C03640=1088.858,407.199,-100.671,177.784,26.140,154.193
C03641=1088.865,407.445,-100.711,177.788,26.148,154.195
C03642=1088.871,407.692,-100.752,177.791,26.157,154.197
C03643=1088.878,407.938,-100.792,177.795,26.166,154.199
C03644=1088.884,408.185,-100.832,177.797,26.175,154.200
C03645=1088.890,408.432,-100.873,177.800,26.183,154.202
C03646=1088.896,408.678,-100.913,177.804,26.192,154.204
C03647=1088.903,408.925,-100.953,177.807,26.201,154.206
C03648=1088.909,409.172,-100.994,177.811,26.210,154.207
C03649=1088.915,409.419,-101.034,177.815,26.219,154.209
C03650=1088.922,409.665,-101.075,177.818,26.227,154.211
C03651=1088.927,409.911,-101.116,177.821,26.236,154.213
C03652=1088.934,410.158,-101.156,177.824,26.245,154.215
C03653=1088.940,410.404,-101.196,177.828,26.254,154.217
C03654=1088.946,410.652,-101.237,177.831,26.263,154.218
C03655=1088.953,410.879,-101.274,177.834,26.272,154.220
C03656=1088.958,411.106,-101.312,177.837,26.280,154.222
C03657=1088.963,411.333,-101.349,177.841,26.288,154.223
C03658=1088.969,411.560,-101.387,177.844,26.297,154.225
C03659=1088.976,411.787,-101.425,177.847,26.305,154.227
C03660=1088.981,412.014,-101.462,177.850,26.313,154.228
C03661=1088.987,412.241,-101.500,177.852,26.322,154.230
C03662=1088.993,412.469,-101.537,177.855,26.330,154.232
C03663=1089.000,412.716,-101.578,177.859,26.339,154.234
C03664=1089.006,412.962,-101.619,177.863,26.349,154.236
C03665=1089.012,413.209,-101.660,177.866,26.358,154.238
C03666=1089.019,413.455,-101.701,177.869,26.368,154.240
C03667=1089.025,413.702,-101.742,177.873,26.377,154.241
C03668=1089.032,413.948,-101.782,177.876,26.386,154.243
C03669=1089.038,414.195,-101.824,177.880,26.395,154.245
C03670=1089.045,414.441,-101.864,177.883,26.405,154.247
C03671=1089.051,414.688,-101.906,177.886,26.414,154.249
C03672=1089.058,414.934,-101.947,177.890,26.423,154.251
C03673=1089.063,415.181,-101.988,177.894,26.433,154.253
C03674=1089.071,415.428,-102.029,177.896,26.442,154.255
C03675=1089.077,415.674,-102.070,177.900,26.452,154.257
C03676=1089.084,415.921,-102.111,177.904,26.462,154.259
C03677=1089.090,416.167,-102.152,177.908,26.471,154.261
C03678=1089.096,416.413,-102.194,177.910,26.481,154.263
C03679=1089.103,416.660,-102.235,177.914,26.490,154.265
C03680=1089.109,416.906,-102.277,177.918,26.500,154.267
C03681=1089.115,417.153,-102.318,177.921,26.510,154.269
C03682=1089.122,417.399,-102.359,177.924,26.520,154.271
C03683=1089.128,417.645,-102.401,177.928,26.529,154.273
C03684=1089.135,417.892,-102.443,177.931,26.539,154.275
C03685=1089.140,418.138,-102.484,177.935,26.549,154.277
C03686=1089.148,418.385,-102.525,177.939,26.559,154.279
C03687=1089.154,418.631,-102.567,177.941,26.569,154.281
C03688=1089.160,418.878,-102.609,177.945,26.579,154.283
C03689=1089.166,419.124,-102.650,177.949,26.589,154.285
C03690=1089.173,419.371,-102.692,177.952,26.599,154.288
C03691=1089.179,419.617,-102.733,177.956,26.609,154.290
C03692=1089.186,419.864,-102.774,177.960,26.619,154.292
C03693=1089.192,420.110,-102.817,177.963,26.630,154.294
C03694=1089.199,420.356,-102.858,177.966,26.639,154.296
C03695=1089.205,420.603,-102.900,177.970,26.649,154.298
C03696=1089.211,420.850,-102.942,177.973,26.660,154.300
C03697=1089.219,421.096,-102.984,177.977,26.670,154.302
C03698=1089.225,421.342,-103.025,177.980,26.680,154.305
C03699=1089.231,421.589,-103.067,177.984,26.691,154.307
C03700=1089.238,421.834,-103.109,177.988,26.701,154.309
C03701=1089.244,422.081,-103.151,177.991,26.711,154.311
C03702=1089.251,422.327,-103.194,177.995,26.722,154.313
C03703=1089.257,422.574,-103.235,177.998,26.732,154.316
C03704=1089.264,422.820,-103.278,178.002,26.743,154.318
C03705=1089.270,423.067,-103.319,178.006,26.753,154.320
C03706=1089.277,423.312,-103.362,178.009,26.764,154.322
C03707=1089.283,423.559,-103.403,178.013,26.775,154.324
C03708=1089.290,423.806,-103.446,178.016,26.785,154.327
C03709=1089.296,424.051,-103.488,178.020,26.796,154.329
C03710=1089.303,424.298,-103.530,178.023,26.807,154.331
C03711=1089.311,424.618,-103.585,178.027,26.820,154.334
C03712=1089.319,424.939,-103.640,178.032,26.834,154.337
C03713=1089.328,425.259,-103.695,178.037,26.849,154.340
C03714=1089.336,425.580,-103.750,178.042,26.863,154.343
C03715=1089.343,425.825,-103.793,178.045,26.874,154.346
C03716=1089.349,426.071,-103.835,178.049,26.884,154.348
C03717=1089.356,426.318,-103.878,178.052,26.895,154.350
C03718=1089.363,426.564,-103.920,178.056,26.906,154.353
C03719=1089.369,426.811,-103.963,178.059,26.918,154.355
C03720=1089.376,427.056,-104.006,178.063,26.928,154.357
C03721=1089.382,427.302,-104.048,178.067,26.940,154.360
C03722=1089.389,427.549,-104.091,178.071,26.951,154.362
C03723=1089.396,427.795,-104.133,178.074,26.962,154.365
C03724=1089.402,428.042,-104.176,178.078,26.973,154.367
C03725=1089.409,428.288,-104.219,178.081,26.985,154.369
C03726=1089.415,428.533,-104.261,178.085,26.996,154.372
C03727=1089.422,428.780,-104.304,178.088,27.007,154.374
C03728=1089.429,429.026,-104.347,178.093,27.019,154.377
C03729=1089.436,429.272,-104.390,178.096,27.030,154.379
C03730=1089.442,429.518,-104.432,178.100,27.041,154.382
C03731=1089.448,429.765,-104.476,178.103,27.053,154.384
C03732=1089.456,430.011,-104.519,178.107,27.065,154.387
C03733=1089.462,430.257,-104.562,178.111,27.076,154.389
C03734=1089.469,430.503,-104.605,178.115,27.088,154.392
C03735=1089.474,430.749,-104.648,178.118,27.099,154.394
C03736=1089.481,430.995,-104.691,178.121,27.111,154.397
C03737=1089.488,431.241,-104.734,178.125,27.123,154.399
C03738=1089.495,431.487,-104.777,178.129,27.135,154.402
C03739=1089.502,431.733,-104.820,178.133,27.146,154.404
C03740=1089.508,431.979,-104.863,178.136,27.158,154.407
C03741=1089.515,432.225,-104.907,178.141,27.171,154.410
C03742=1089.521,432.472,-104.950,178.144,27.182,154.412
C03743=1089.528,432.717,-104.993,178.147,27.194,154.415
C03744=1089.535,432.963,-105.037,178.151,27.206,154.418
C03745=1089.542,433.210,-105.079,178.155,27.218,154.420
C03746=1089.548,433.456,-105.123,178.159,27.231,154.423
C03747=1089.554,433.702,-105.167,178.162,27.242,154.426
C03748=1089.562,433.947,-105.210,178.166,27.255,154.428
C03749=1089.568,434.194,-105.253,178.170,27.267,154.431
C03750=1089.575,434.441,-105.298,178.173,27.279,154.434
C03751=1089.586,434.835,-105.368,178.180,27.300,154.438
C03752=1089.596,435.230,-105.438,178.186,27.319,154.442
C03753=1089.607,435.626,-105.508,178.192,27.339,154.447
C03754=1089.617,436.021,-105.578,178.198,27.359,154.451
C03755=1089.624,436.266,-105.622,178.202,27.372,154.454
C03756=1089.631,436.512,-105.666,178.205,27.385,154.457
C03757=1089.638,436.759,-105.710,178.209,27.398,154.460
C03758=1089.645,437.004,-105.754,178.213,27.410,154.463
C03759=1089.651,437.250,-105.798,178.217,27.423,154.465
C03760=1089.658,437.496,-105.841,178.220,27.436,154.468
C03761=1089.664,437.742,-105.886,178.225,27.449,154.471
C03762=1089.671,437.988,-105.930,178.228,27.461,154.474
C03763=1089.680,438.310,-105.987,178.234,27.479,154.478
C03764=1089.689,438.630,-106.045,178.238,27.495,154.481
C03765=1089.698,438.952,-106.103,178.244,27.512,154.485
C03766=1089.707,439.273,-106.161,178.248,27.529,154.489
C03767=1089.714,439.519,-106.204,178.252,27.543,154.492
C03768=1089.720,439.764,-106.249,178.256,27.556,154.495
C03769=1089.728,440.010,-106.293,178.260,27.569,154.498
C03770=1089.735,440.256,-106.337,178.264,27.583,154.501
C03771=1089.742,440.501,-106.382,178.268,27.596,154.504
C03772=1089.748,440.748,-106.426,178.272,27.609,154.507
C03773=1089.755,440.993,-106.471,178.275,27.623,154.510
C03774=1089.762,441.240,-106.515,178.279,27.637,154.513
C03775=1089.768,441.485,-106.560,178.284,27.650,154.516
C03776=1089.775,441.731,-106.604,178.287,27.664,154.519
C03777=1089.782,441.977,-106.649,178.291,27.677,154.522
C03778=1089.789,442.222,-106.694,178.296,27.691,154.525
C03779=1089.797,442.468,-106.739,178.299,27.705,154.529
C03780=1089.803,442.714,-106.783,178.303,27.719,154.532
C03781=1089.810,442.959,-106.827,178.307,27.733,154.535
C03782=1089.816,443.206,-106.873,178.311,27.747,154.538
C03783=1089.823,443.451,-106.917,178.315,27.761,154.541
C03784=1089.830,443.697,-106.962,178.319,27.775,154.544
C03785=1089.837,443.943,-107.007,178.323,27.789,154.547
C03786=1089.844,444.189,-107.052,178.327,27.803,154.551
C03787=1089.851,444.434,-107.098,178.331,27.817,154.554
C03788=1089.858,444.680,-107.143,178.335,27.832,154.557
C03789=1089.865,444.925,-107.187,178.338,27.846,154.560
C03790=1089.872,445.171,-107.232,178.342,27.860,154.564
C03791=1089.879,445.418,-107.278,178.345,27.874,154.567
C03792=1089.886,445.662,-107.323,178.348,27.888,154.570
C03793=1089.893,445.908,-107.368,178.351,27.903,154.574
C03794=1089.899,446.154,-107.413,178.354,27.917,154.577
C03795=1089.907,446.399,-107.459,178.356,27.931,154.580
C03796=1089.913,446.646,-107.504,178.358,27.945,154.584
C03797=1089.920,446.891,-107.549,178.361,27.959,154.587
C03798=1089.928,447.137,-107.594,178.363,27.973,154.591
C03799=1089.934,447.383,-107.640,178.364,27.987,154.594
C03800=1089.941,447.628,-107.685,178.366,28.001,154.597
C03801=1089.948,447.874,-107.731,178.367,28.015,154.601
C03802=1089.956,448.119,-107.776,178.368,28.030,154.604
C03803=1089.962,448.366,-107.822,178.370,28.043,154.608
C03804=1089.969,448.611,-107.867,178.371,28.058,154.611
C03805=1089.976,448.857,-107.913,178.372,28.071,154.615
C03806=1089.983,449.102,-107.958,178.373,28.086,154.618
C03807=1089.990,449.347,-108.004,178.373,28.100,154.622
C03808=1089.997,449.593,-108.050,178.374,28.114,154.625
C03809=1090.004,449.838,-108.094,178.374,28.128,154.629
C03810=1090.015,450.084,-108.139,178.374,28.140,154.632
C03811=1089.633,450.077,-108.327,178.332,28.336,154.686
C03812=1089.623,449.830,-108.284,178.331,28.323,154.682
C03813=1089.615,449.585,-108.238,178.330,28.310,154.679
C03814=1089.609,449.340,-108.192,178.330,28.295,154.675
C03815=1089.602,449.095,-108.147,178.329,28.281,154.672
C03816=1089.594,448.849,-108.102,178.329,28.267,154.669
C03817=1089.587,448.603,-108.056,178.327,28.253,154.665
C03818=1089.580,448.358,-108.010,178.326,28.239,154.662
C03819=1089.573,448.111,-107.964,178.325,28.225,154.658
C03820=1089.566,447.867,-107.919,178.324,28.211,154.655
C03821=1089.559,447.620,-107.874,178.322,28.197,154.651
C03822=1089.552,447.375,-107.828,178.320,28.183,154.648
C03823=1089.545,447.128,-107.782,178.318,28.169,154.644
C03824=1089.538,446.884,-107.737,178.316,28.154,154.641
C03825=1089.532,446.637,-107.692,178.314,28.140,154.637
C03826=1089.524,446.392,-107.646,178.311,28.126,154.634
C03827=1089.517,446.146,-107.601,178.309,28.111,154.631
C03828=1089.510,445.901,-107.555,178.306,28.097,154.627
C03829=1089.503,445.655,-107.510,178.303,28.083,154.624
C03830=1089.497,445.409,-107.465,178.300,28.069,154.621
C03831=1089.489,445.164,-107.419,178.296,28.055,154.617
C03832=1089.482,444.918,-107.374,178.293,28.040,154.614
C03833=1089.475,444.672,-107.330,178.289,28.027,154.611
C03834=1089.468,444.426,-107.284,178.285,28.012,154.607
C03835=1089.462,444.181,-107.239,178.281,27.998,154.604
C03836=1089.454,443.935,-107.194,178.277,27.984,154.601
C03837=1089.448,443.690,-107.150,178.273,27.969,154.598
C03838=1089.441,443.443,-107.104,178.269,27.955,154.595
C03839=1089.434,443.198,-107.060,178.264,27.941,154.591
C03840=1089.427,442.952,-107.015,178.261,27.927,154.588
C03841=1089.420,442.707,-106.970,178.257,27.913,154.585
C03842=1089.413,442.460,-106.925,178.252,27.899,154.582
C03843=1089.406,442.215,-106.881,178.249,27.886,154.579
C03844=1089.400,441.969,-106.835,178.245,27.872,154.576
C03845=1089.393,441.723,-106.790,178.240,27.858,154.573
C03846=1089.385,441.477,-106.745,178.237,27.844,154.570
C03847=1089.379,441.232,-106.701,178.233,27.831,154.567
C03848=1089.372,440.986,-106.657,178.229,27.817,154.563
C03849=1089.365,440.740,-106.612,178.225,27.803,154.560
C03850=1089.358,440.495,-106.568,178.220,27.790,154.557
C03851=1089.351,440.249,-106.523,178.217,27.777,154.554
C03852=1089.345,440.003,-106.479,178.213,27.763,154.551
C03853=1089.338,439.757,-106.434,178.209,27.750,154.548
C03854=1089.331,439.511,-106.390,178.205,27.736,154.545
C03855=1089.324,439.265,-106.345,178.201,27.723,154.542
C03856=1089.315,438.957,-106.290,178.196,27.707,154.539
C03857=1089.307,438.648,-106.235,178.191,27.690,154.535
C03858=1089.298,438.340,-106.179,178.186,27.674,154.531
C03859=1089.290,438.031,-106.124,178.181,27.658,154.528
C03860=1089.283,437.785,-106.080,178.177,27.645,154.525
C03861=1089.275,437.540,-106.036,178.174,27.632,154.522
C03862=1089.269,437.294,-105.992,178.169,27.619,154.519
C03863=1089.262,437.048,-105.948,178.166,27.606,154.516
C03864=1089.255,436.801,-105.904,178.162,27.593,154.514
C03865=1089.249,436.556,-105.859,178.158,27.581,154.511
C03866=1089.241,436.310,-105.816,178.154,27.568,154.508
C03867=1089.235,436.064,-105.772,178.150,27.555,154.505
C03868=1089.229,435.818,-105.728,178.146,27.543,154.502
C03869=1089.222,435.572,-105.684,178.142,27.530,154.500
C03870=1089.214,435.326,-105.641,178.139,27.518,154.497
C03871=1089.208,435.080,-105.597,178.135,27.505,154.494
C03872=1089.202,434.834,-105.553,178.131,27.493,154.491
C03873=1089.195,434.588,-105.509,178.127,27.480,154.489
C03874=1089.188,434.342,-105.466,178.124,27.468,154.486
C03875=1089.181,434.096,-105.422,178.119,27.456,154.483
C03876=1089.175,433.850,-105.378,178.116,27.443,154.480
C03877=1089.168,433.605,-105.335,178.112,27.431,154.478
C03878=1089.161,433.359,-105.291,178.108,27.419,154.475
C03879=1089.155,433.112,-105.248,178.104,27.407,154.472
C03880=1089.149,432.866,-105.204,178.101,27.394,154.470
C03881=1089.141,432.620,-105.160,178.096,27.382,154.467
C03882=1089.135,432.373,-105.117,178.093,27.371,154.464
C03883=1089.128,432.127,-105.074,178.089,27.358,154.462
C03884=1089.121,431.882,-105.030,178.085,27.346,154.459
C03885=1089.115,431.635,-104.988,178.081,27.335,154.457
C03886=1089.108,431.389,-104.944,178.078,27.323,154.454
C03887=1089.101,431.143,-104.901,178.074,27.311,154.451
C03888=1089.094,430.897,-104.858,178.071,27.299,154.449
C03889=1089.088,430.651,-104.815,178.066,27.287,154.446
C03890=1089.081,430.405,-104.772,178.063,27.276,154.444
C03891=1089.075,430.158,-104.729,178.059,27.264,154.441
C03892=1089.068,429.913,-104.685,178.056,27.253,154.439
C03893=1089.062,429.667,-104.643,178.051,27.241,154.436
C03894=1089.055,429.421,-104.600,178.048,27.230,154.434
C03895=1089.048,429.175,-104.557,178.044,27.218,154.431
C03896=1089.042,428.928,-104.514,178.041,27.206,154.429
C03897=1089.035,428.682,-104.471,178.037,27.195,154.426
C03898=1089.028,428.436,-104.428,178.033,27.184,154.424
C03899=1089.022,428.190,-104.385,178.030,27.172,154.421
C03900=1089.015,427.944,-104.342,178.025,27.161,154.419
C03901=1089.008,427.697,-104.300,178.022,27.150,154.417
C03902=1089.001,427.451,-104.257,178.018,27.139,154.414
C03903=1088.996,427.205,-104.214,178.015,27.128,154.412
C03904=1088.989,426.959,-104.172,178.011,27.116,154.409
C03905=1088.982,426.713,-104.129,178.007,27.106,154.407
C03906=1088.975,426.466,-104.087,178.004,27.094,154.405
C03907=1088.968,426.220,-104.044,178.000,27.083,154.402
C03908=1088.962,425.984,-104.004,177.996,27.073,154.400
C03909=1088.956,425.750,-103.963,177.993,27.062,154.398
C03910=1088.950,425.514,-103.922,177.989,27.052,154.396
C03911=1088.944,425.279,-103.882,177.986,27.042,154.393
C03912=1088.937,425.044,-103.841,177.983,27.031,154.391
C03913=1088.931,424.809,-103.801,177.979,27.021,154.389
C03914=1088.925,424.572,-103.760,177.975,27.010,154.387
C03915=1088.919,424.337,-103.719,177.972,27.000,154.384
C03916=1088.912,424.091,-103.677,177.969,26.989,154.382
C03917=1088.906,423.845,-103.635,177.965,26.979,154.380
C03918=1088.899,423.598,-103.593,177.962,26.968,154.378
C03919=1088.893,423.353,-103.551,177.958,26.958,154.375
C03920=1088.886,423.106,-103.508,177.954,26.947,154.373
C03921=1088.879,422.859,-103.466,177.951,26.936,154.371
C03922=1088.873,422.614,-103.424,177.947,26.925,154.369
C03923=1088.867,422.367,-103.382,177.943,26.915,154.366
C03924=1088.860,422.121,-103.340,177.940,26.904,154.364
C03925=1088.854,421.874,-103.298,177.936,26.894,154.362
C03926=1088.847,421.628,-103.256,177.932,26.884,154.360
C03927=1088.840,421.381,-103.214,177.929,26.873,154.358
C03928=1088.834,421.136,-103.172,177.925,26.863,154.355
C03929=1088.828,420.889,-103.130,177.921,26.853,154.353
C03930=1088.821,420.643,-103.089,177.918,26.843,154.351
C03931=1088.814,420.397,-103.047,177.915,26.832,154.349
C03932=1088.807,420.150,-103.005,177.911,26.822,154.347
C03933=1088.802,419.903,-102.963,177.907,26.812,154.345
C03934=1088.795,419.657,-102.921,177.904,26.802,154.343
C03935=1088.789,419.411,-102.879,177.900,26.792,154.341
C03936=1088.781,419.164,-102.838,177.896,26.781,154.338
C03937=1088.775,418.918,-102.797,177.894,26.772,154.336
C03938=1088.769,418.671,-102.755,177.890,26.762,154.334
C03939=1088.763,418.425,-102.713,177.886,26.752,154.332
C03940=1088.756,418.178,-102.672,177.882,26.742,154.330
C03941=1088.750,417.932,-102.631,177.879,26.732,154.328
C03942=1088.743,417.685,-102.589,177.876,26.722,154.326
C03943=1088.737,417.439,-102.547,177.872,26.712,154.324
C03944=1088.730,417.181,-102.503,177.869,26.702,154.322
C03945=1088.723,416.924,-102.461,177.865,26.691,154.320
C03946=1088.717,416.666,-102.417,177.861,26.681,154.317
C03947=1088.710,416.408,-102.373,177.858,26.671,154.315
C03948=1088.704,416.162,-102.332,177.854,26.661,154.313
C03949=1088.698,415.915,-102.292,177.850,26.652,154.311
C03950=1088.691,415.669,-102.250,177.847,26.643,154.309
C03951=1088.684,415.423,-102.209,177.844,26.633,154.307
C03952=1088.678,415.176,-102.167,177.840,26.623,154.305
C03953=1088.671,414.930,-102.126,177.837,26.614,154.303
C03954=1088.665,414.682,-102.085,177.833,26.604,154.301
C03955=1088.658,414.436,-102.044,177.829,26.595,154.300
C03956=1088.652,414.190,-102.002,177.826,26.585,154.298
C03957=1088.645,413.943,-101.962,177.823,26.576,154.296
C03958=1088.639,413.697,-101.921,177.819,26.567,154.294
C03959=1088.632,413.450,-101.880,177.816,26.557,154.292
C03960=1088.626,413.204,-101.839,177.812,26.548,154.290
C03961=1088.620,412.957,-101.798,177.809,26.539,154.288
C03962=1088.613,412.710,-101.757,177.806,26.530,154.286
C03963=1088.607,412.464,-101.716,177.802,26.520,154.284
C03964=1088.602,412.241,-101.680,177.799,26.512,154.283
C03965=1088.595,412.020,-101.643,177.796,26.504,154.281
C03966=1088.589,411.798,-101.606,177.793,26.495,154.279
C03967=1088.584,411.575,-101.570,177.790,26.487,154.278
C03968=1088.578,411.353,-101.533,177.787,26.479,154.276
C03969=1088.572,411.131,-101.496,177.784,26.471,154.274
C03970=1088.567,410.909,-101.460,177.780,26.463,154.273
C03971=1088.561,410.687,-101.422,177.777,26.455,154.271
C03972=1088.555,410.440,-101.382,177.774,26.445,154.269
C03973=1088.548,410.194,-101.341,177.771,26.437,154.267
C03974=1088.542,409.948,-101.301,177.767,26.427,154.265
C03975=1088.535,409.700,-101.260,177.764,26.419,154.264
C03976=1088.529,409.454,-101.220,177.760,26.410,154.262
C03977=1088.523,409.207,-101.179,177.757,26.401,154.260
C03978=1088.517,408.961,-101.138,177.753,26.392,154.258
C03979=1088.510,408.715,-101.098,177.750,26.383,154.256
C03980=1088.505,408.468,-101.057,177.747,26.374,154.255
C03981=1088.498,408.221,-101.017,177.744,26.365,154.253
C03982=1088.492,407.975,-100.977,177.740,26.357,154.251
C03983=1088.486,407.727,-100.936,177.737,26.348,154.249
C03984=1088.479,407.481,-100.896,177.733,26.339,154.247
C03985=1088.473,407.234,-100.856,177.730,26.331,154.246
C03986=1088.467,406.988,-100.816,177.726,26.321,154.244
C03987=1088.460,406.741,-100.775,177.723,26.313,154.242
C03988=1088.455,406.494,-100.735,177.720,26.305,154.241
C03989=1088.448,406.248,-100.695,177.716,26.296,154.239
C03990=1088.442,406.001,-100.654,177.713,26.288,154.237
C03991=1088.435,405.755,-100.614,177.710,26.278,154.235
C03992=1088.429,405.508,-100.575,177.707,26.271,154.234
C03993=1088.423,405.261,-100.535,177.704,26.262,154.232
C03994=1088.416,405.014,-100.494,177.700,26.254,154.230
C03995=1088.410,404.767,-100.454,177.697,26.245,154.229
C03996=1088.403,404.520,-100.415,177.693,26.236,154.227
C03997=1088.397,404.274,-100.374,177.690,26.228,154.225
C03998=1088.391,404.027,-100.334,177.687,26.220,154.224
C03999=1088.384,403.781,-100.294,177.683,26.211,154.222
C04000=1088.378,403.534,-100.255,177.680,26.203,154.220
C04001=1088.372,403.287,-100.215,177.677,26.195,154.219
C04002=1088.366,403.040,-100.175,177.673,26.187,154.217
C04003=1088.359,402.794,-100.135,177.670,26.178,154.215
C04004=1088.353,402.547,-100.095,177.667,26.171,154.214
C04005=1088.347,402.300,-100.055,177.663,26.162,154.212
C04006=1088.341,402.054,-100.016,177.660,26.154,154.211
C04007=1088.335,401.807,-99.976,177.657,26.146,154.209
C04008=1088.329,401.560,-99.936,177.653,26.138,154.207
C04009=1088.322,401.314,-99.897,177.650,26.130,154.206
C04010=1088.316,401.066,-99.858,177.647,26.122,154.204
C04011=1088.309,400.820,-99.818,177.644,26.114,154.203
C04012=1088.303,400.573,-99.778,177.640,26.106,154.201
C04013=1088.297,400.326,-99.738,177.637,26.098,154.200
C04014=1088.291,400.079,-99.699,177.634,26.090,154.198
C04015=1088.285,399.833,-99.660,177.631,26.082,154.196
C04016=1088.278,399.587,-99.620,177.627,26.074,154.195
C04017=1088.272,399.339,-99.581,177.624,26.066,154.193
C04018=1088.266,399.092,-99.541,177.621,26.058,154.192
C04019=1088.260,398.845,-99.502,177.618,26.050,154.190
C04020=1088.255,398.618,-99.466,177.615,26.043,154.189
C04021=1088.249,398.392,-99.429,177.611,26.036,154.187
C04022=1088.243,398.164,-99.393,177.608,26.029,154.186
C04023=1088.237,397.938,-99.357,177.606,26.022,154.185
C04024=1088.231,397.711,-99.321,177.603,26.015,154.183
C04025=1088.225,397.483,-99.285,177.600,26.007,154.182
C04026=1088.220,397.256,-99.249,177.596,26.000,154.181
C04027=1088.214,397.029,-99.213,177.593,25.993,154.179
C04028=1088.208,396.782,-99.174,177.590,25.985,154.178
C04029=1088.202,396.535,-99.134,177.587,25.978,154.176
C04030=1088.195,396.288,-99.096,177.584,25.970,154.175
C04031=1088.190,396.041,-99.056,177.581,25.963,154.173
C04032=1088.183,395.795,-99.018,177.578,25.955,154.172
C04033=1088.177,395.547,-98.978,177.574,25.947,154.170
C04034=1088.171,395.301,-98.939,177.570,25.940,154.169
C04035=1088.164,395.054,-98.900,177.567,25.932,154.167
C04036=1088.158,394.807,-98.861,177.564,25.925,154.166
C04037=1088.152,394.561,-98.822,177.561,25.917,154.165
C04038=1088.146,394.314,-98.783,177.558,25.910,154.163
C04039=1088.139,394.067,-98.744,177.555,25.902,154.162
C04040=1088.134,393.820,-98.706,177.552,25.895,154.160
C04041=1088.127,393.573,-98.667,177.548,25.888,154.159
C04042=1088.121,393.326,-98.628,177.545,25.880,154.157
C04043=1088.115,393.080,-98.589,177.541,25.873,154.156
C04044=1088.109,392.832,-98.551,177.538,25.866,154.155
C04045=1088.103,392.586,-98.512,177.535,25.858,154.153
C04046=1088.096,392.339,-98.473,177.532,25.851,154.152
C04047=1088.091,392.092,-98.435,177.529,25.844,154.150
C04048=1088.084,391.845,-98.396,177.526,25.836,154.149
C04049=1088.077,391.598,-98.357,177.522,25.829,154.148
C04050=1088.072,391.352,-98.319,177.519,25.822,154.146
C04051=1088.065,391.105,-98.280,177.516,25.815,154.145
C04052=1088.060,390.858,-98.242,177.512,25.807,154.144
C04053=1088.053,390.611,-98.203,177.509,25.800,154.142
C04054=1088.046,390.364,-98.164,177.506,25.793,154.141
C04055=1088.041,390.117,-98.126,177.502,25.786,154.140
C04056=1088.034,389.870,-98.087,177.499,25.779,154.138
C04057=1088.028,389.624,-98.049,177.496,25.772,154.137
C04058=1088.022,389.376,-98.011,177.493,25.765,154.136
C04059=1088.015,389.130,-97.973,177.490,25.758,154.134
C04060=1088.009,388.883,-97.935,177.486,25.751,154.133
C04061=1088.003,388.636,-97.896,177.483,25.744,154.132
C04062=1087.997,388.389,-97.858,177.480,25.737,154.131
C04063=1087.991,388.142,-97.820,177.477,25.730,154.129
C04064=1087.985,387.896,-97.781,177.474,25.723,154.128
C04065=1087.978,387.648,-97.743,177.470,25.716,154.127
C04066=1087.972,387.402,-97.705,177.467,25.709,154.125
C04067=1087.966,387.155,-97.667,177.464,25.703,154.124
C04068=1087.960,386.908,-97.628,177.461,25.696,154.123
C04069=1087.954,386.661,-97.590,177.458,25.689,154.122
C04070=1087.948,386.414,-97.552,177.454,25.682,154.120
C04071=1087.942,386.167,-97.515,177.451,25.675,154.119
C04072=1087.936,385.921,-97.476,177.448,25.668,154.118
C04073=1087.929,385.673,-97.438,177.445,25.661,154.116
C04074=1087.923,385.427,-97.400,177.441,25.655,154.115
C04075=1087.918,385.180,-97.362,177.438,25.648,154.114
C04076=1087.912,384.959,-97.328,177.435,25.641,154.113
C04077=1087.907,384.738,-97.294,177.432,25.636,154.112
C04078=1087.901,384.519,-97.261,177.430,25.630,154.111
C04079=1087.896,384.297,-97.227,177.426,25.623,154.110
C04080=1087.891,384.077,-97.193,177.424,25.618,154.108
C04081=1087.886,383.857,-97.159,177.421,25.611,154.107
C04082=1087.879,383.637,-97.126,177.418,25.606,154.106
C04083=1087.874,383.417,-97.091,177.416,25.600,154.105
C04084=1087.868,383.170,-97.054,177.412,25.593,154.104
C04085=1087.862,382.922,-97.016,177.409,25.586,154.103
C04086=1087.856,382.675,-96.978,177.406,25.580,154.102
C04087=1087.850,382.429,-96.941,177.403,25.573,154.100
C04088=1087.844,382.181,-96.903,177.399,25.566,154.099
C04089=1087.838,381.934,-96.865,177.396,25.560,154.098
C04090=1087.831,381.688,-96.828,177.393,25.554,154.097
C04091=1087.826,381.441,-96.790,177.389,25.547,154.096
C04092=1087.819,381.193,-96.753,177.386,25.540,154.095
C04093=1087.813,380.946,-96.715,177.383,25.534,154.093
C04094=1087.807,380.700,-96.678,177.380,25.528,154.092
C04095=1087.801,380.453,-96.641,177.377,25.521,154.091
C04096=1087.795,380.205,-96.602,177.374,25.515,154.090
C04097=1087.789,379.958,-96.565,177.370,25.509,154.089
C04098=1087.783,379.711,-96.528,177.367,25.502,154.088
C04099=1087.777,379.465,-96.490,177.364,25.496,154.087
C04100=1087.771,379.218,-96.453,177.360,25.489,154.085
C04101=1087.764,378.970,-96.415,177.357,25.483,154.084
C04102=1087.758,378.723,-96.378,177.355,25.477,154.083
C04103=1087.752,378.476,-96.341,177.351,25.471,154.082
C04104=1087.746,378.229,-96.303,177.348,25.464,154.081
C04105=1087.741,377.982,-96.266,177.345,25.458,154.080
C04106=1087.734,377.735,-96.229,177.342,25.451,154.079
C04107=1087.728,377.487,-96.192,177.338,25.445,154.077
C04108=1087.722,377.241,-96.154,177.335,25.439,154.076
C04109=1087.716,376.994,-96.118,177.332,25.433,154.075
C04110=1087.710,376.747,-96.080,177.329,25.427,154.074
C04111=1087.704,376.500,-96.043,177.326,25.420,154.073
C04112=1087.698,376.252,-96.006,177.322,25.414,154.072
C04113=1087.692,376.006,-95.969,177.319,25.408,154.071
C04114=1087.686,375.758,-95.932,177.317,25.402,154.070
C04115=1087.680,375.511,-95.895,177.313,25.396,154.069
C04116=1087.674,375.265,-95.857,177.310,25.389,154.068
C04117=1087.668,375.017,-95.820,177.306,25.383,154.067
C04118=1087.662,374.770,-95.784,177.303,25.377,154.066
C04119=1087.656,374.523,-95.747,177.301,25.371,154.064
C04120=1087.651,374.276,-95.709,177.297,25.365,154.063
C04121=1087.644,374.029,-95.673,177.294,25.358,154.062
C04122=1087.638,373.781,-95.635,177.291,25.353,154.061
C04123=1087.632,373.534,-95.599,177.287,25.347,154.060
C04124=1087.625,373.287,-95.562,177.285,25.341,154.059
C04125=1087.620,373.039,-95.525,177.281,25.335,154.058
C04126=1087.613,372.792,-95.489,177.278,25.329,154.057
C04127=1087.608,372.546,-95.451,177.275,25.323,154.056
C04128=1087.601,372.299,-95.415,177.272,25.317,154.055
C04129=1087.595,372.052,-95.378,177.269,25.311,154.054
C04130=1087.589,371.804,-95.341,177.265,25.305,154.053
C04131=1087.583,371.557,-95.305,177.262,25.299,154.052
C04132=1087.573,371.144,-95.244,177.257,25.289,154.050
C04133=1087.563,370.731,-95.182,177.251,25.279,154.049
C04134=1087.553,370.318,-95.121,177.247,25.270,154.047
C04135=1087.543,369.906,-95.060,177.241,25.260,154.045
C04136=1087.536,369.659,-95.024,177.238,25.254,154.044
C04137=1087.531,369.411,-94.988,177.234,25.248,154.043
C04138=1087.525,369.164,-94.951,177.231,25.242,154.042
C04139=1087.518,368.917,-94.915,177.229,25.237,154.041
C04140=1087.513,368.669,-94.878,177.225,25.231,154.040
C04141=1087.507,368.422,-94.842,177.222,25.225,154.039
C04142=1087.501,368.175,-94.806,177.219,25.220,154.038
C04143=1087.495,367.928,-94.769,177.216,25.214,154.037
C04144=1087.489,367.681,-94.732,177.212,25.208,154.036
C04145=1087.483,367.433,-94.697,177.210,25.202,154.035
C04146=1087.477,367.186,-94.660,177.206,25.197,154.034
C04147=1087.471,366.939,-94.623,177.203,25.191,154.034
C04148=1087.466,366.692,-94.588,177.200,25.186,154.033
C04149=1087.459,366.445,-94.551,177.197,25.179,154.032
C04150=1087.453,366.197,-94.516,177.194,25.174,154.031
C04151=1087.448,365.950,-94.479,177.191,25.168,154.030
C04152=1087.442,365.702,-94.443,177.188,25.163,154.029
C04153=1087.436,365.456,-94.407,177.184,25.157,154.028
C04154=1087.430,365.208,-94.371,177.182,25.151,154.027
C04155=1087.424,364.961,-94.335,177.178,25.146,154.026
C04156=1087.418,364.713,-94.299,177.175,25.140,154.025
C04157=1087.411,364.466,-94.262,177.172,25.135,154.024
C04158=1087.405,364.219,-94.227,177.169,25.129,154.023
C04159=1087.400,363.972,-94.190,177.165,25.124,154.022
C04160=1087.394,363.724,-94.154,177.163,25.118,154.021
C04161=1087.388,363.477,-94.119,177.159,25.113,154.020
C04162=1087.382,363.229,-94.082,177.156,25.107,154.020
C04163=1087.376,362.982,-94.046,177.153,25.102,154.019
C04164=1087.370,362.735,-94.011,177.150,25.096,154.018
C04165=1087.364,362.488,-93.975,177.146,25.091,154.017
C04166=1087.358,362.240,-93.939,177.143,25.086,154.016
C04167=1087.352,361.992,-93.903,177.140,25.080,154.015
C04168=1087.347,361.745,-93.868,177.137,25.075,154.014
C04169=1087.339,361.499,-93.832,177.134,25.069,154.013
C04170=1087.333,361.251,-93.796,177.130,25.064,154.013
C04171=1087.327,361.003,-93.760,177.128,25.059,154.012
C04172=1087.322,360.756,-93.725,177.124,25.053,154.011
C04173=1087.316,360.509,-93.689,177.122,25.048,154.010
C04174=1087.310,360.262,-93.653,177.118,25.042,154.009
C04175=1087.304,360.015,-93.618,177.115,25.037,154.008
C04176=1087.298,359.767,-93.582,177.112,25.032,154.007
C04177=1087.292,359.519,-93.546,177.109,25.026,154.006
C04178=1087.287,359.272,-93.511,177.106,25.021,154.006
C04179=1087.280,359.025,-93.476,177.102,25.016,154.005
C04180=1087.274,358.777,-93.440,177.099,25.010,154.004
C04181=1087.268,358.530,-93.404,177.096,25.005,154.003
C04182=1087.262,358.283,-93.369,177.093,25.000,154.002
C04183=1087.256,358.035,-93.333,177.090,24.995,154.001
C04184=1087.247,357.638,-93.277,177.084,24.986,154.000
C04185=1087.237,357.241,-93.220,177.080,24.978,153.999
C04186=1087.227,356.843,-93.163,177.075,24.970,153.997
C04187=1087.218,356.446,-93.106,177.069,24.961,153.996
C04188=1087.212,356.199,-93.071,177.067,24.956,153.995
C04189=1087.206,355.952,-93.035,177.063,24.951,153.994
C04190=1087.200,355.705,-93.001,177.061,24.946,153.993
C04191=1087.195,355.457,-92.966,177.057,24.941,153.993
C04192=1087.189,355.209,-92.930,177.054,24.936,153.992
C04193=1087.182,354.962,-92.895,177.051,24.930,153.991
C04194=1087.176,354.715,-92.859,177.048,24.926,153.990
C04195=1087.171,354.467,-92.825,177.045,24.920,153.989
C04196=1087.164,354.220,-92.790,177.042,24.915,153.989
C04197=1087.159,353.973,-92.754,177.038,24.910,153.988
C04198=1087.153,353.724,-92.719,177.036,24.905,153.987
C04199=1087.147,353.478,-92.684,177.032,24.900,153.986
C04200=1087.141,353.230,-92.649,177.030,24.895,153.985
C04201=1087.136,352.982,-92.614,177.026,24.890,153.985
C04202=1087.129,352.735,-92.579,177.023,24.885,153.984
C04203=1087.124,352.487,-92.544,177.020,24.880,153.983
C04204=1087.117,352.240,-92.509,177.017,24.875,153.982
C04205=1087.112,351.992,-92.474,177.013,24.870,153.982
C04206=1087.105,351.745,-92.439,177.011,24.865,153.981
C04207=1087.100,351.498,-92.405,177.007,24.860,153.980
C04208=1087.094,351.250,-92.370,177.005,24.855,153.979
C04209=1087.088,351.003,-92.335,177.001,24.850,153.979
C04210=1087.082,350.755,-92.300,176.998,24.845,153.978
C04211=1087.077,350.508,-92.265,176.995,24.840,153.977
C04212=1087.070,350.260,-92.231,176.992,24.836,153.976
C04213=1087.065,350.013,-92.195,176.988,24.830,153.975
C04214=1087.058,349.765,-92.161,176.986,24.826,153.975
C04215=1087.053,349.518,-92.126,176.982,24.820,153.974
C04216=1087.046,349.270,-92.091,176.979,24.816,153.973
C04217=1087.040,349.022,-92.057,176.976,24.811,153.972
C04218=1087.035,348.775,-92.022,176.973,24.806,153.972
C04219=1087.029,348.527,-91.987,176.970,24.801,153.971
C04220=1087.023,348.280,-91.953,176.967,24.796,153.970
C04221=1087.017,348.032,-91.918,176.964,24.792,153.969
C04222=1087.011,347.785,-91.884,176.961,24.786,153.969
C04223=1087.006,347.538,-91.849,176.958,24.782,153.968
C04224=1086.999,347.290,-91.814,176.954,24.777,153.967
C04225=1086.993,347.042,-91.780,176.951,24.772,153.967
C04226=1086.988,346.794,-91.745,176.948,24.767,153.966
C04227=1086.982,346.547,-91.711,176.945,24.762,153.965
C04228=1086.976,346.300,-91.677,176.942,24.758,153.964
C04229=1086.970,346.051,-91.642,176.939,24.753,153.964
C04230=1086.964,345.805,-91.607,176.936,24.748,153.963
C04231=1086.958,345.557,-91.573,176.932,24.743,153.962
C04232=1086.952,345.309,-91.538,176.930,24.739,153.962
C04233=1086.947,345.062,-91.504,176.927,24.734,153.961
C04234=1086.941,344.814,-91.470,176.923,24.729,153.960
C04235=1086.934,344.566,-91.436,176.921,24.724,153.959
C04236=1086.925,344.172,-91.382,176.916,24.717,153.958
C04237=1086.916,343.778,-91.327,176.911,24.710,153.957
C04238=1086.906,343.383,-91.272,176.906,24.702,153.956
C04239=1086.897,342.989,-91.218,176.901,24.695,153.955
C04240=1086.891,342.741,-91.184,176.897,24.690,153.954
C04241=1086.885,342.494,-91.150,176.895,24.685,153.954
C04242=1086.880,342.246,-91.115,176.892,24.681,153.953
C04243=1086.874,341.999,-91.081,176.888,24.676,153.952
C04244=1086.868,341.751,-91.048,176.885,24.672,153.952
C04245=1086.862,341.503,-91.013,176.883,24.667,153.951
C04246=1086.856,341.255,-90.979,176.879,24.662,153.950
C04247=1086.850,341.008,-90.945,176.876,24.658,153.950
C04248=1086.844,340.760,-90.912,176.873,24.653,153.949
C04249=1086.839,340.513,-90.878,176.870,24.648,153.948
C04250=1086.832,340.265,-90.844,176.867,24.644,153.948
C04251=1086.827,340.017,-90.810,176.863,24.640,153.947
C04252=1086.821,339.770,-90.776,176.861,24.635,153.946
C04253=1086.815,339.522,-90.742,176.858,24.631,153.946
C04254=1086.809,339.275,-90.709,176.854,24.626,153.945
C04255=1086.803,339.027,-90.674,176.851,24.621,153.944
C04256=1086.797,338.779,-90.640,176.849,24.617,153.944
C04257=1086.791,338.531,-90.607,176.845,24.612,153.943
C04258=1086.786,338.284,-90.573,176.842,24.608,153.942
C04259=1086.780,338.036,-90.540,176.839,24.604,153.942
C04260=1086.774,337.789,-90.505,176.836,24.599,153.941
C04261=1086.768,337.540,-90.472,176.833,24.594,153.940
C04262=1086.762,337.293,-90.438,176.830,24.590,153.940
C04263=1086.757,337.045,-90.404,176.827,24.585,153.939
C04264=1086.751,336.798,-90.370,176.824,24.581,153.938
C04265=1086.745,336.550,-90.337,176.821,24.577,153.938
C04266=1086.739,336.303,-90.304,176.818,24.572,153.937
C04267=1086.733,336.055,-90.270,176.814,24.568,153.937
C04268=1086.727,335.807,-90.237,176.812,24.564,153.936
C04269=1086.721,335.559,-90.202,176.809,24.559,153.935
C04270=1086.715,335.311,-90.169,176.805,24.555,153.935
C04271=1086.709,335.064,-90.136,176.802,24.550,153.934
C04272=1086.703,334.816,-90.102,176.799,24.546,153.933
C04273=1086.698,334.568,-90.069,176.796,24.541,153.933
C04274=1086.692,334.321,-90.036,176.793,24.537,153.932
C04275=1086.686,334.073,-90.002,176.790,24.533,153.932
C04276=1086.680,333.826,-89.969,176.788,24.528,153.931
C04277=1086.674,333.578,-89.936,176.784,24.524,153.930
C04278=1086.669,333.330,-89.902,176.781,24.519,153.930
C04279=1086.663,333.083,-89.868,176.778,24.515,153.929
C04280=1086.657,332.835,-89.835,176.775,24.511,153.928
C04281=1086.651,332.587,-89.802,176.772,24.507,153.928
C04282=1086.646,332.339,-89.769,176.769,24.502,153.927
C04283=1086.640,332.091,-89.735,176.766,24.498,153.927
C04284=1086.634,331.844,-89.703,176.763,24.494,153.926
C04285=1086.628,331.596,-89.669,176.760,24.489,153.925
C04286=1086.622,331.348,-89.635,176.757,24.485,153.925
C04287=1086.616,331.101,-89.602,176.754,24.481,153.924
C04288=1086.606,330.700,-89.549,176.749,24.475,153.923
C04289=1086.596,330.300,-89.496,176.744,24.467,153.922
C04290=1086.587,329.900,-89.442,176.739,24.461,153.922
C04291=1086.577,329.500,-89.389,176.733,24.454,153.921
C04292=1086.571,329.252,-89.356,176.731,24.450,153.920
C04293=1086.566,329.004,-89.323,176.728,24.446,153.920
C04294=1086.559,328.757,-89.290,176.725,24.442,153.919
C04295=1086.554,328.509,-89.257,176.722,24.438,153.918
C04296=1086.547,328.261,-89.224,176.718,24.433,153.918
C04297=1086.541,328.013,-89.192,176.715,24.429,153.917
C04298=1086.536,327.765,-89.159,176.713,24.425,153.917
C04299=1086.530,327.518,-89.126,176.710,24.421,153.916
C04300=1086.524,327.270,-89.093,176.706,24.417,153.916
C04301=1086.518,327.022,-89.060,176.703,24.412,153.915
C04302=1086.511,326.774,-89.027,176.700,24.408,153.914
C04303=1086.507,326.527,-88.995,176.698,24.404,153.914
C04304=1086.501,326.279,-88.962,176.695,24.400,153.913
C04305=1086.495,326.031,-88.929,176.692,24.396,153.913
C04306=1086.489,325.784,-88.896,176.688,24.392,153.912
C04307=1086.483,325.535,-88.864,176.685,24.388,153.912
C04308=1086.477,325.287,-88.831,176.682,24.384,153.911
C04309=1086.471,325.040,-88.798,176.679,24.380,153.911
C04310=1086.465,324.792,-88.766,176.677,24.376,153.910
C04311=1086.460,324.544,-88.733,176.673,24.371,153.910
C04312=1086.454,324.297,-88.700,176.670,24.367,153.909
C04313=1086.448,324.049,-88.668,176.667,24.363,153.908
C04314=1086.442,323.801,-88.635,176.664,24.359,153.908
C04315=1086.436,323.552,-88.603,176.661,24.355,153.907
C04316=1086.430,323.305,-88.570,176.659,24.351,153.907
C04317=1086.425,323.058,-88.537,176.655,24.347,153.906
C04318=1086.419,322.809,-88.505,176.652,24.343,153.906
C04319=1086.413,322.562,-88.472,176.649,24.339,153.905
C04320=1086.407,322.313,-88.440,176.646,24.335,153.905
C04321=1086.402,322.066,-88.407,176.643,24.331,153.904
C04322=1086.396,321.818,-88.375,176.640,24.327,153.904
C04323=1086.389,321.571,-88.343,176.638,24.323,153.903
C04324=1086.384,321.322,-88.310,176.634,24.319,153.903
C04325=1086.379,321.075,-88.278,176.631,24.314,153.902
C04326=1086.372,320.827,-88.246,176.628,24.310,153.901
C04327=1086.367,320.578,-88.213,176.625,24.306,153.901
C04328=1086.361,320.332,-88.181,176.622,24.303,153.901
C04329=1086.355,320.083,-88.148,176.619,24.299,153.900
C04330=1086.349,319.835,-88.116,176.617,24.295,153.899
C04331=1086.343,319.588,-88.084,176.614,24.291,153.899
C04332=1086.339,319.340,-88.051,176.610,24.286,153.898
C04333=1086.333,319.092,-88.019,176.607,24.282,153.898
C04334=1086.327,318.845,-87.987,176.604,24.279,153.897
C04335=1086.321,318.596,-87.955,176.601,24.275,153.897
C04336=1086.316,318.348,-87.922,176.598,24.271,153.896
C04337=1086.310,318.100,-87.891,176.596,24.267,153.896
C04338=1086.304,317.853,-87.858,176.593,24.263,153.895
C04339=1086.298,317.605,-87.826,176.590,24.259,153.895
C04340=1086.289,317.198,-87.774,176.585,24.252,153.894
C04341=1086.280,316.790,-87.721,176.580,24.246,153.893
C04342=1086.270,316.384,-87.668,176.574,24.239,153.892
C04343=1086.261,315.977,-87.615,176.570,24.233,153.891
C04344=1086.256,315.729,-87.583,176.567,24.229,153.891
C04345=1086.250,315.481,-87.551,176.564,24.225,153.890
C04346=1086.244,315.234,-87.520,176.561,24.221,153.890
C04347=1086.238,314.986,-87.488,176.558,24.217,153.889
C04348=1086.233,314.738,-87.456,176.555,24.213,153.889
C04349=1086.227,314.490,-87.424,176.552,24.209,153.888
C04350=1086.221,314.242,-87.392,176.549,24.205,153.888
C04351=1086.215,313.994,-87.360,176.546,24.202,153.887
C04352=1086.209,313.746,-87.329,176.543,24.198,153.887
C04353=1086.203,313.498,-87.297,176.540,24.194,153.886
C04354=1086.197,313.250,-87.265,176.537,24.190,153.886
C04355=1086.191,313.002,-87.233,176.534,24.187,153.886
C04356=1086.185,312.755,-87.202,176.531,24.183,153.885
C04357=1086.179,312.507,-87.170,176.529,24.179,153.885
C04358=1086.174,312.258,-87.139,176.526,24.176,153.884
C04359=1086.168,312.010,-87.107,176.523,24.172,153.884
C04360=1086.161,311.763,-87.076,176.519,24.167,153.883
C04361=1086.156,311.515,-87.044,176.516,24.164,153.883
C04362=1086.150,311.267,-87.012,176.513,24.160,153.882
C04363=1086.144,311.020,-86.981,176.510,24.156,153.882
C04364=1086.138,310.771,-86.950,176.507,24.153,153.881
C04365=1086.133,310.523,-86.918,176.504,24.149,153.881
C04366=1086.127,310.275,-86.886,176.501,24.145,153.880
C04367=1086.121,310.028,-86.855,176.498,24.142,153.880
C04368=1086.115,309.780,-86.823,176.495,24.138,153.880
C04369=1086.110,309.532,-86.792,176.492,24.134,153.879
C04370=1086.103,309.284,-86.760,176.489,24.130,153.879
C04371=1086.098,309.036,-86.729,176.486,24.127,153.878
C04372=1086.092,308.787,-86.697,176.484,24.123,153.878
C04373=1086.086,308.540,-86.666,176.481,24.119,153.877
C04374=1086.080,308.292,-86.634,176.478,24.116,153.877
C04375=1086.074,308.044,-86.604,176.475,24.112,153.876
C04376=1086.068,307.796,-86.572,176.472,24.108,153.876
C04377=1086.063,307.548,-86.540,176.469,24.104,153.875
C04378=1086.057,307.300,-86.510,176.466,24.101,153.875
C04379=1086.051,307.052,-86.478,176.463,24.097,153.875
C04380=1086.046,306.804,-86.447,176.460,24.093,153.874
C04381=1086.040,306.557,-86.416,176.457,24.090,153.874
C04382=1086.034,306.308,-86.385,176.454,24.086,153.873
C04383=1086.028,306.061,-86.354,176.451,24.083,153.873
C04384=1086.022,305.812,-86.322,176.448,24.078,153.872
C04385=1086.016,305.565,-86.291,176.445,24.075,153.872
C04386=1086.011,305.317,-86.260,176.442,24.071,153.872
C04387=1086.005,305.069,-86.228,176.439,24.067,153.871
C04388=1085.999,304.821,-86.198,176.436,24.063,153.871
C04389=1085.994,304.573,-86.166,176.433,24.060,153.870
C04390=1085.988,304.325,-86.136,176.430,24.056,153.870
C04391=1085.982,304.077,-86.104,176.427,24.053,153.869
C04392=1085.973,303.673,-86.054,176.422,24.047,153.869
C04393=1085.963,303.269,-86.004,176.417,24.040,153.868
C04394=1085.954,302.865,-85.953,176.413,24.035,153.867
C04395=1085.945,302.461,-85.903,176.408,24.028,153.866
C04396=1085.939,302.213,-85.871,176.405,24.025,153.866
C04397=1085.934,301.965,-85.840,176.402,24.021,153.866
C04398=1085.928,301.717,-85.810,176.399,24.018,153.865
C04399=1085.923,301.469,-85.779,176.396,24.014,153.865
C04400=1085.916,301.221,-85.748,176.393,24.010,153.864
C04401=1085.911,300.973,-85.717,176.391,24.007,153.864
C04402=1085.905,300.725,-85.686,176.388,24.003,153.863
C04403=1085.900,300.477,-85.655,176.385,24.000,153.863
C04404=1085.894,300.229,-85.625,176.382,23.996,153.862
C04405=1085.889,299.982,-85.593,176.379,23.992,153.862
C04406=1085.882,299.733,-85.563,176.376,23.989,153.862
C04407=1085.877,299.485,-85.532,176.373,23.985,153.861
C04408=1085.872,299.237,-85.501,176.370,23.981,153.861
C04409=1085.866,298.989,-85.471,176.367,23.978,153.860
C04410=1085.861,298.741,-85.440,176.364,23.974,153.860
C04411=1085.855,298.493,-85.410,176.362,23.970,153.859
C04412=1085.850,298.245,-85.379,176.359,23.967,153.859
C04413=1085.843,297.997,-85.348,176.356,23.963,153.859
C04414=1085.837,297.749,-85.318,176.353,23.960,153.858
C04415=1085.832,297.501,-85.287,176.350,23.956,153.858
C04416=1085.827,297.253,-85.256,176.347,23.953,153.857
C04417=1085.821,297.005,-85.226,176.344,23.949,153.857
C04418=1085.815,296.757,-85.196,176.341,23.945,153.857
C04419=1085.809,296.509,-85.165,176.338,23.942,153.856
C04420=1085.803,296.261,-85.134,176.335,23.938,153.856
C04421=1085.798,296.013,-85.104,176.332,23.935,153.855
C04422=1085.792,295.765,-85.073,176.330,23.931,153.855
C04423=1085.786,295.517,-85.043,176.327,23.928,153.854
C04424=1085.780,295.269,-85.013,176.324,23.924,153.854
C04425=1085.775,295.021,-84.983,176.321,23.921,153.854
C04426=1085.768,294.772,-84.952,176.318,23.918,153.853
C04427=1085.763,294.524,-84.921,176.315,23.914,153.853
C04428=1085.757,294.276,-84.891,176.312,23.910,153.853
C04429=1085.752,294.028,-84.861,176.309,23.907,153.852
C04430=1085.746,293.780,-84.831,176.306,23.903,153.852
C04431=1085.740,293.532,-84.801,176.303,23.900,153.851
C04432=1085.734,293.285,-84.770,176.300,23.896,153.851
C04433=1085.729,293.036,-84.741,176.297,23.893,153.851
C04434=1085.723,292.788,-84.710,176.295,23.890,153.850
C04435=1085.717,292.540,-84.680,176.292,23.886,153.850
C04436=1085.711,292.293,-84.649,176.289,23.882,153.849
C04437=1085.706,292.044,-84.620,176.286,23.879,153.849
C04438=1085.699,291.796,-84.589,176.283,23.876,153.849
C04439=1085.694,291.548,-84.559,176.280,23.872,153.848
C04440=1085.688,291.299,-84.529,176.277,23.869,153.848
C04441=1085.682,291.052,-84.499,176.274,23.865,153.847
C04442=1085.677,290.803,-84.469,176.271,23.861,153.847
C04443=1085.671,290.555,-84.439,176.269,23.859,153.847
C04444=1085.662,290.165,-84.391,176.264,23.853,153.846
C04445=1085.653,289.776,-84.344,176.259,23.847,153.846
C04446=1085.645,289.386,-84.298,176.255,23.842,153.845
C04447=1085.635,288.995,-84.250,176.250,23.837,153.844
C04448=1085.629,288.747,-84.220,176.247,23.833,153.844
C04449=1085.624,288.499,-84.190,176.244,23.830,153.844
C04450=1085.618,288.251,-84.161,176.242,23.827,153.843
C04451=1085.612,288.003,-84.131,176.239,23.823,153.843
C04452=1085.606,287.755,-84.101,176.236,23.820,153.843
C04453=1085.600,287.507,-84.071,176.233,23.816,153.842
C04454=1085.595,287.258,-84.041,176.230,23.813,153.842
C04455=1085.589,287.010,-84.012,176.227,23.810,153.841
C04456=1085.583,286.762,-83.982,176.224,23.806,153.841
C04457=1085.578,286.515,-83.953,176.222,23.803,153.841
C04458=1085.572,286.266,-83.923,176.219,23.800,153.840
C04459=1085.566,286.018,-83.893,176.216,23.796,153.840
C04460=1085.560,285.770,-83.864,176.213,23.793,153.839
C04461=1085.555,285.522,-83.834,176.210,23.789,153.839
C04462=1085.549,285.274,-83.804,176.207,23.786,153.839
C04463=1085.543,285.026,-83.774,176.204,23.782,153.838
C04464=1085.537,284.777,-83.745,176.202,23.780,153.838
C04465=1085.532,284.529,-83.715,176.199,23.776,153.838
C04466=1085.526,284.281,-83.686,176.196,23.772,153.837
C04467=1085.520,284.033,-83.655,176.193,23.769,153.837
C04468=1085.514,283.785,-83.626,176.190,23.766,153.837
C04469=1085.509,283.537,-83.597,176.187,23.762,153.836
C04470=1085.504,283.288,-83.568,176.185,23.759,153.836
C04471=1085.498,283.040,-83.538,176.182,23.756,153.835
C04472=1085.492,282.792,-83.509,176.179,23.753,153.835
C04473=1085.486,282.543,-83.479,176.176,23.749,153.835
C04474=1085.481,282.296,-83.449,176.173,23.745,153.834
C04475=1085.475,282.048,-83.420,176.170,23.742,153.834
C04476=1085.469,281.800,-83.391,176.168,23.739,153.834
C04477=1085.464,281.551,-83.361,176.165,23.735,153.833
C04478=1085.458,281.303,-83.332,176.162,23.732,153.833
C04479=1085.452,281.055,-83.302,176.159,23.729,153.833
C04480=1085.447,280.806,-83.273,176.156,23.726,153.832
C04481=1085.441,280.559,-83.244,176.154,23.722,153.832
C04482=1085.435,280.310,-83.214,176.150,23.719,153.832
C04483=1085.429,280.062,-83.185,176.148,23.716,153.831
C04484=1085.424,279.814,-83.156,176.145,23.712,153.831
C04485=1085.417,279.566,-83.127,176.142,23.709,153.831
C04486=1085.413,279.317,-83.098,176.139,23.706,153.830
C04487=1085.407,279.069,-83.069,176.136,23.703,153.830
C04488=1085.401,278.821,-83.039,176.133,23.699,153.829
C04489=1085.395,278.573,-83.010,176.130,23.696,153.829
C04490=1085.389,278.324,-82.981,176.127,23.692,153.829
C04491=1085.384,278.077,-82.952,176.125,23.689,153.828
C04492=1085.378,277.828,-82.922,176.122,23.686,153.828
C04493=1085.372,277.580,-82.894,176.119,23.683,153.828
C04494=1085.367,277.331,-82.864,176.116,23.679,153.827
C04495=1085.361,277.084,-82.836,176.113,23.676,153.827
C04496=1085.352,276.703,-82.791,176.110,23.671,153.826
C04497=1085.343,276.323,-82.746,176.105,23.666,153.826
C04498=1085.334,275.943,-82.702,176.101,23.661,153.825
C04499=1085.326,275.562,-82.658,176.096,23.656,153.825
C04500=1085.320,275.314,-82.629,176.093,23.653,153.825
C04501=1085.314,275.066,-82.600,176.091,23.650,153.824
C04502=1085.308,274.817,-82.571,176.088,23.646,153.824
C04503=1085.303,274.569,-82.542,176.085,23.643,153.824
C04504=1085.297,274.321,-82.513,176.082,23.639,153.823
C04505=1085.292,274.072,-82.484,176.080,23.637,153.823
C04506=1085.286,273.825,-82.455,176.077,23.633,153.823
C04507=1085.280,273.576,-82.427,176.074,23.630,153.822
C04508=1085.274,273.328,-82.398,176.071,23.626,153.822
C04509=1085.269,273.079,-82.369,176.069,23.624,153.822
C04510=1085.263,272.831,-82.340,176.065,23.620,153.821
C04511=1085.257,272.583,-82.311,176.062,23.617,153.821
C04512=1085.252,272.335,-82.283,176.059,23.614,153.821
C04513=1085.246,272.087,-82.254,176.057,23.610,153.820
C04514=1085.240,271.838,-82.225,176.054,23.607,153.820
C04515=1085.235,271.590,-82.198,176.051,23.604,153.820
C04516=1085.229,271.342,-82.168,176.048,23.601,153.819
C04517=1085.223,271.093,-82.140,176.046,23.598,153.819
C04518=1085.218,270.845,-82.111,176.043,23.595,153.819
C04519=1085.212,270.596,-82.083,176.040,23.591,153.818
C04520=1085.206,270.349,-82.054,176.037,23.588,153.818
C04521=1085.200,270.100,-82.026,176.035,23.585,153.818
C04522=1085.195,269.851,-81.997,176.032,23.582,153.817
C04523=1085.189,269.604,-81.968,176.029,23.578,153.817
C04524=1085.183,269.355,-81.940,176.026,23.575,153.817
C04525=1085.178,269.107,-81.912,176.024,23.572,153.816
C04526=1085.172,268.859,-81.883,176.021,23.569,153.816
C04527=1085.166,268.610,-81.854,176.018,23.565,153.816
C04528=1085.160,268.362,-81.826,176.015,23.563,153.815
C04529=1085.154,268.114,-81.797,176.012,23.559,153.815
C04530=1085.149,267.866,-81.769,176.009,23.556,153.815
C04531=1085.143,267.617,-81.741,176.006,23.553,153.814
C04532=1085.138,267.368,-81.712,176.004,23.550,153.814
C04533=1085.132,267.120,-81.684,176.001,23.546,153.814
C04534=1085.126,266.872,-81.655,175.998,23.543,153.813
C04535=1085.121,266.624,-81.627,175.995,23.540,153.813
C04536=1085.115,266.375,-81.599,175.993,23.537,153.813
C04537=1085.110,266.127,-81.571,175.990,23.534,153.812
C04538=1085.104,265.878,-81.543,175.987,23.531,153.812
C04539=1085.098,265.630,-81.515,175.985,23.527,153.812
C04540=1085.092,265.382,-81.486,175.982,23.524,153.811
C04541=1085.087,265.134,-81.458,175.979,23.521,153.811
C04542=1085.081,264.885,-81.429,175.977,23.518,153.811
C04543=1085.075,264.637,-81.401,175.974,23.515,153.810
C04544=1085.069,264.388,-81.373,175.971,23.512,153.810
C04545=1085.064,264.140,-81.345,175.968,23.508,153.810
C04546=1085.058,263.892,-81.317,175.965,23.505,153.809
C04547=1085.052,263.644,-81.289,175.962,23.502,153.809
C04548=1085.043,263.266,-81.247,175.958,23.497,153.809
C04549=1085.034,262.888,-81.204,175.954,23.493,153.808
C04550=1085.025,262.511,-81.161,175.949,23.488,153.808
C04551=1085.016,262.133,-81.119,175.946,23.483,153.807
C04552=1085.011,261.885,-81.091,175.943,23.480,153.807
C04553=1085.005,261.636,-81.063,175.940,23.477,153.807
C04554=1084.999,261.389,-81.035,175.937,23.474,153.807
C04555=1084.993,261.140,-81.007,175.935,23.471,153.806
C04556=1084.988,260.892,-80.979,175.931,23.468,153.806
C04557=1084.982,260.643,-80.951,175.929,23.465,153.806
C04558=1084.976,260.395,-80.924,175.926,23.462,153.805
C04559=1084.971,260.147,-80.896,175.923,23.459,153.805
C04560=1084.965,259.898,-80.868,175.921,23.456,153.805
C04561=1084.959,259.650,-80.840,175.918,23.452,153.804
C04562=1084.953,259.401,-80.812,175.915,23.449,153.804
C04563=1084.948,259.153,-80.785,175.913,23.446,153.804
C04564=1084.941,258.904,-80.757,175.910,23.443,153.804
C04565=1084.936,258.656,-80.729,175.907,23.440,153.803
C04566=1084.930,258.408,-80.701,175.904,23.437,153.803
C04567=1084.924,258.159,-80.674,175.902,23.434,153.803
C04568=1084.919,257.911,-80.646,175.898,23.430,153.802
C04569=1084.913,257.662,-80.618,175.896,23.428,153.802
C04570=1084.907,257.414,-80.591,175.893,23.425,153.802
C04571=1084.902,257.166,-80.563,175.890,23.421,153.801
C04572=1084.896,256.917,-80.535,175.888,23.418,153.801
C04573=1084.890,256.669,-80.508,175.885,23.415,153.801
C04574=1084.885,256.421,-80.480,175.882,23.412,153.801
C04575=1084.879,256.172,-80.452,175.880,23.409,153.800
C04576=1084.873,255.924,-80.425,175.877,23.406,153.800
C04577=1084.867,255.676,-80.397,175.874,23.403,153.800
C04578=1084.861,255.427,-80.370,175.872,23.400,153.799
C04579=1084.856,255.179,-80.342,175.869,23.396,153.799
C04580=1084.851,254.930,-80.315,175.866,23.394,153.799
C04581=1084.844,254.681,-80.287,175.863,23.391,153.798
C04582=1084.839,254.433,-80.260,175.860,23.387,153.798
C04583=1084.833,254.185,-80.233,175.858,23.384,153.798
C04584=1084.827,253.936,-80.205,175.855,23.381,153.797
C04585=1084.822,253.688,-80.177,175.852,23.378,153.797
C04586=1084.816,253.439,-80.151,175.850,23.375,153.797
C04587=1084.811,253.191,-80.123,175.847,23.372,153.797
C04588=1084.804,252.942,-80.096,175.844,23.368,153.796
C04589=1084.799,252.694,-80.068,175.842,23.366,153.796
C04590=1084.793,252.446,-80.041,175.839,23.362,153.796
C04591=1084.788,252.197,-80.014,175.837,23.360,153.795
C04592=1084.783,251.949,-79.986,175.833,23.356,153.795
C04593=1084.777,251.700,-79.959,175.831,23.353,153.795
C04594=1084.772,251.451,-79.932,175.828,23.350,153.794
C04595=1084.765,251.204,-79.904,175.825,23.347,153.794
C04596=1084.760,250.955,-79.877,175.823,23.344,153.794
C04597=1084.754,250.706,-79.850,175.820,23.340,153.793
C04598=1084.749,250.458,-79.822,175.817,23.337,153.793
C04599=1084.743,250.209,-79.795,175.815,23.335,153.793
C04600=1084.735,249.829,-79.753,175.811,23.330,153.792
C04601=1084.726,249.449,-79.712,175.807,23.325,153.792
C04602=1084.718,249.068,-79.671,175.802,23.320,153.791
C04603=1084.709,248.688,-79.629,175.799,23.315,153.791
C04604=1084.704,248.440,-79.602,175.796,23.312,153.791
C04605=1084.698,248.191,-79.575,175.794,23.310,153.790
C04606=1084.693,247.943,-79.548,175.790,23.306,153.790
C04607=1084.687,247.695,-79.521,175.788,23.303,153.790
C04608=1084.682,247.446,-79.493,175.785,23.300,153.789
C04609=1084.676,247.197,-79.466,175.782,23.297,153.789
C04610=1084.670,246.949,-79.440,175.780,23.294,153.789
C04611=1084.665,246.700,-79.412,175.777,23.291,153.789
C04612=1084.659,246.452,-79.386,175.774,23.287,153.788
C04613=1084.653,246.203,-79.359,175.772,23.284,153.788
C04614=1084.648,245.955,-79.332,175.769,23.281,153.788
C04615=1084.642,245.706,-79.305,175.767,23.279,153.787
C04616=1084.636,245.457,-79.278,175.764,23.275,153.787
C04617=1084.630,245.209,-79.252,175.762,23.273,153.787
C04618=1084.625,244.960,-79.224,175.759,23.269,153.787
C04619=1084.619,244.712,-79.198,175.756,23.266,153.786
C04620=1084.614,244.464,-79.171,175.753,23.263,153.786
C04621=1084.609,244.215,-79.144,175.750,23.260,153.786
C04622=1084.603,243.967,-79.117,175.748,23.257,153.785
C04623=1084.597,243.718,-79.090,175.745,23.254,153.785
C04624=1084.591,243.470,-79.064,175.743,23.251,153.785
C04625=1084.585,243.221,-79.037,175.740,23.248,153.784
C04626=1084.580,242.973,-79.010,175.737,23.244,153.784
C04627=1084.575,242.724,-78.983,175.735,23.242,153.784
C04628=1084.569,242.476,-78.957,175.732,23.238,153.784
C04629=1084.563,242.226,-78.930,175.730,23.236,153.783
C04630=1084.557,241.978,-78.904,175.727,23.232,153.783
C04631=1084.551,241.730,-78.877,175.724,23.230,153.783
C04632=1084.546,241.481,-78.850,175.721,23.227,153.782
C04633=1084.540,241.233,-78.824,175.719,23.224,153.782
C04634=1084.534,240.984,-78.798,175.716,23.221,153.782
C04635=1084.528,240.736,-78.771,175.713,23.217,153.782
C04636=1084.523,240.487,-78.745,175.711,23.215,153.781
C04637=1084.517,240.239,-78.718,175.708,23.211,153.781
C04638=1084.511,239.990,-78.692,175.706,23.209,153.781
C04639=1084.506,239.741,-78.665,175.703,23.206,153.780
C04640=1084.501,239.493,-78.638,175.701,23.203,153.780
C04641=1084.494,239.245,-78.612,175.697,23.200,153.780
C04642=1084.489,238.996,-78.586,175.695,23.197,153.780
C04643=1084.483,238.747,-78.559,175.692,23.194,153.779
C04644=1084.477,238.499,-78.533,175.690,23.190,153.779
C04645=1084.472,238.250,-78.507,175.687,23.187,153.779
C04646=1084.466,238.002,-78.480,175.685,23.184,153.778
C04647=1084.460,237.753,-78.454,175.682,23.181,153.778
C04648=1084.455,237.504,-78.428,175.680,23.179,153.778
C04649=1084.449,237.256,-78.401,175.677,23.175,153.778
C04650=1084.443,237.007,-78.375,175.675,23.173,153.777
C04651=1084.438,236.759,-78.348,175.672,23.169,153.777
C04652=1084.429,236.372,-78.308,175.668,23.165,153.777
C04653=1084.420,235.985,-78.267,175.664,23.160,153.776
C04654=1084.411,235.598,-78.226,175.660,23.156,153.776
C04655=1084.402,235.210,-78.185,175.655,23.151,153.775
C04656=1084.397,234.961,-78.159,175.653,23.148,153.775
C04657=1084.391,234.713,-78.133,175.650,23.145,153.775
C04658=1084.386,234.465,-78.107,175.648,23.142,153.774
C04659=1084.381,234.216,-78.080,175.645,23.138,153.774
C04660=1084.375,233.967,-78.054,175.643,23.136,153.774
C04661=1084.369,233.719,-78.028,175.640,23.132,153.773
C04662=1084.363,233.470,-78.002,175.638,23.130,153.773
C04663=1084.358,233.221,-77.977,175.635,23.126,153.773
C04664=1084.352,232.973,-77.950,175.632,23.124,153.773
C04665=1084.346,232.724,-77.924,175.629,23.120,153.772
C04666=1084.342,232.476,-77.898,175.627,23.118,153.772
C04667=1084.335,232.228,-77.872,175.624,23.114,153.772
C04668=1084.330,231.979,-77.846,175.622,23.112,153.772
C04669=1084.324,231.730,-77.820,175.619,23.109,153.771
C04670=1084.318,231.481,-77.794,175.617,23.106,153.771
C04671=1084.313,231.232,-77.768,175.614,23.103,153.771
C04672=1084.307,230.984,-77.743,175.612,23.100,153.770
C04673=1084.302,230.735,-77.717,175.609,23.097,153.770
C04674=1084.296,230.487,-77.690,175.606,23.094,153.770
C04675=1084.290,230.238,-77.665,175.604,23.090,153.769
C04676=1084.284,229.989,-77.639,175.601,23.087,153.769
C04677=1084.279,229.740,-77.613,175.598,23.085,153.769
C04678=1084.273,229.492,-77.588,175.596,23.082,153.769
C04679=1084.268,229.244,-77.561,175.593,23.079,153.769
C04680=1084.261,228.995,-77.536,175.591,23.076,153.768
C04681=1084.256,228.746,-77.510,175.589,23.073,153.768
C04682=1084.250,228.497,-77.484,175.586,23.070,153.768
C04683=1084.245,228.250,-77.459,175.584,23.067,153.767
C04684=1084.239,228.001,-77.433,175.580,23.064,153.767
C04685=1084.233,227.752,-77.408,175.578,23.061,153.767
C04686=1084.228,227.503,-77.382,175.575,23.058,153.767
C04687=1084.222,227.255,-77.355,175.573,23.055,153.766
C04688=1084.216,227.007,-77.330,175.570,23.052,153.766
C04689=1084.211,226.758,-77.305,175.568,23.049,153.766
C04690=1084.205,226.509,-77.279,175.565,23.046,153.765
C04691=1084.199,226.260,-77.253,175.563,23.043,153.765
C04692=1084.194,226.012,-77.228,175.561,23.040,153.765
C04693=1084.188,225.763,-77.202,175.558,23.037,153.764
C04694=1084.182,225.514,-77.177,175.556,23.034,153.764
C04695=1084.176,225.265,-77.151,175.553,23.031,153.764
C04696=1084.171,225.017,-77.126,175.550,23.028,153.764
C04697=1084.165,224.768,-77.100,175.547,23.025,153.763
C04698=1084.159,224.520,-77.075,175.545,23.022,153.763
C04699=1084.155,224.271,-77.050,175.542,23.019,153.763
C04700=1084.148,224.022,-77.025,175.540,23.016,153.763
C04701=1084.143,223.773,-76.999,175.538,23.013,153.762
C04702=1084.137,223.525,-76.974,175.535,23.010,153.762
C04703=1084.132,223.276,-76.948,175.533,23.007,153.762
C04704=1084.123,222.880,-76.908,175.528,23.002,153.761
C04705=1084.114,222.485,-76.867,175.525,22.998,153.761
C04706=1084.105,222.089,-76.827,175.520,22.993,153.760
C04707=1084.096,221.693,-76.787,175.516,22.989,153.760
C04708=1084.090,221.445,-76.762,175.513,22.985,153.760
C04709=1084.085,221.197,-76.736,175.511,22.983,153.759
C04710=1084.079,220.948,-76.711,175.509,22.980,153.759
C04711=1084.073,220.699,-76.686,175.506,22.977,153.759
C04712=1084.068,220.450,-76.660,175.504,22.974,153.759
C04713=1084.062,220.202,-76.635,175.501,22.971,153.758
C04714=1084.056,219.953,-76.610,175.499,22.968,153.758
C04715=1084.050,219.704,-76.586,175.497,22.965,153.758
C04716=1084.045,219.455,-76.560,175.494,22.962,153.758
C04717=1084.039,219.207,-76.534,175.491,22.959,153.757
C04718=1084.033,218.958,-76.510,175.488,22.956,153.757
C04719=1084.027,218.709,-76.485,175.486,22.953,153.757
C04720=1084.022,218.461,-76.459,175.484,22.950,153.756
C04721=1084.016,218.212,-76.434,175.481,22.947,153.756
C04722=1084.011,217.964,-76.410,175.479,22.944,153.756
C04723=1084.005,217.715,-76.385,175.476,22.941,153.756
C04724=1083.999,217.466,-76.359,175.474,22.938,153.755
C04725=1083.994,217.218,-76.334,175.472,22.936,153.755
C04726=1083.988,216.968,-76.309,175.469,22.932,153.755
C04727=1083.982,216.720,-76.284,175.467,22.930,153.754
C04728=1083.977,216.471,-76.259,175.464,22.926,153.754
C04729=1083.971,216.223,-76.234,175.461,22.924,153.754
C04730=1083.966,215.974,-76.210,175.459,22.921,153.754
C04731=1083.960,215.726,-76.185,175.456,22.918,153.753
C04732=1083.954,215.476,-76.160,175.454,22.915,153.753
C04733=1083.948,215.228,-76.135,175.452,22.912,153.753
C04734=1083.943,214.979,-76.110,175.449,22.909,153.753
C04735=1083.938,214.731,-76.085,175.447,22.906,153.752
C04736=1083.932,214.481,-76.060,175.444,22.903,153.752
C04737=1083.926,214.233,-76.036,175.442,22.900,153.752
C04738=1083.920,213.984,-76.011,175.440,22.897,153.751
C04739=1083.916,213.735,-75.986,175.437,22.894,153.751
C04740=1083.909,213.487,-75.960,175.434,22.891,153.751
C04741=1083.904,213.238,-75.936,175.432,22.888,153.750
C04742=1083.898,212.989,-75.912,175.429,22.885,153.750
C04743=1083.893,212.741,-75.887,175.427,22.882,153.750
C04744=1083.887,212.492,-75.862,175.424,22.879,153.750
C04745=1083.881,212.243,-75.838,175.422,22.876,153.749
C04746=1083.875,211.994,-75.812,175.420,22.873,153.749
C04747=1083.870,211.746,-75.788,175.417,22.870,153.749
C04748=1083.864,211.496,-75.763,175.415,22.867,153.749
C04749=1083.859,211.248,-75.739,175.413,22.864,153.748
C04750=1083.853,211.000,-75.714,175.410,22.861,153.748
C04751=1083.847,210.751,-75.690,175.407,22.858,153.748
C04752=1083.842,210.502,-75.665,175.405,22.856,153.747
C04753=1083.836,210.253,-75.641,175.402,22.852,153.747
C04754=1083.830,210.005,-75.616,175.400,22.850,153.747
C04755=1083.825,209.755,-75.591,175.398,22.847,153.747
C04756=1083.816,209.364,-75.553,175.393,22.842,153.746
C04757=1083.807,208.972,-75.514,175.390,22.838,153.746
C04758=1083.798,208.581,-75.476,175.386,22.833,153.745
C04759=1083.789,208.189,-75.437,175.382,22.828,153.745
C04760=1083.766,207.159,-75.338,175.294,22.782,153.748
C04761=1083.761,206.910,-75.314,175.292,22.780,153.748
C04762=1083.755,206.662,-75.290,175.289,22.778,153.748
C04763=1083.749,206.412,-75.266,175.287,22.776,153.747
C04764=1083.744,206.164,-75.242,175.284,22.774,153.747
C04765=1083.738,205.915,-75.218,175.282,22.772,153.747
C04766=1083.733,205.666,-75.195,175.279,22.770,153.747
C04767=1083.727,205.418,-75.171,175.276,22.768,153.747
C04768=1083.721,205.169,-75.147,175.274,22.766,153.747
C04769=1083.716,204.919,-75.123,175.271,22.764,153.747
C04770=1083.710,204.671,-75.099,175.269,22.762,153.747
C04771=1083.704,204.423,-75.075,175.267,22.760,153.747
C04772=1083.699,204.173,-75.051,175.264,22.758,153.747
C04773=1083.693,203.925,-75.028,175.262,22.756,153.747
C04774=1083.688,203.676,-75.003,175.258,22.754,153.747
C04775=1083.682,203.428,-74.981,175.256,22.752,153.747
C04776=1083.676,203.178,-74.956,175.254,22.750,153.747
C04777=1083.671,202.929,-74.932,175.251,22.748,153.747
C04778=1083.665,202.681,-74.909,175.249,22.746,153.747
C04779=1083.660,202.432,-74.885,175.246,22.744,153.746
C04780=1083.654,202.183,-74.862,175.244,22.742,153.746
C04781=1083.649,201.934,-74.838,175.241,22.740,153.746
C04782=1083.643,201.686,-74.814,175.239,22.738,153.746
C04783=1083.637,201.436,-74.791,175.236,22.736,153.746
C04784=1083.632,201.188,-74.767,175.233,22.734,153.746
C04785=1083.626,200.939,-74.744,175.231,22.732,153.746
C04786=1083.620,200.690,-74.720,175.228,22.730,153.746
C04787=1083.615,200.441,-74.697,175.226,22.728,153.746
C04788=1083.609,200.193,-74.673,175.223,22.726,153.746
C04789=1083.604,199.944,-74.649,175.221,22.725,153.746
C04790=1083.597,199.695,-74.625,175.218,22.723,153.746
C04791=1083.591,199.446,-74.602,175.216,22.720,153.746
C04792=1083.586,199.197,-74.578,175.214,22.719,153.746
C04793=1083.580,198.948,-74.555,175.211,22.717,153.746
C04794=1083.575,198.700,-74.532,175.209,22.715,153.746
C04795=1083.569,198.451,-74.508,175.206,22.713,153.746
C04796=1083.564,198.202,-74.485,175.203,22.711,153.746
C04797=1083.558,197.953,-74.462,175.200,22.709,153.746
C04798=1083.553,197.705,-74.438,175.198,22.707,153.746
C04799=1083.547,197.456,-74.415,175.196,22.705,153.746
C04800=1083.541,197.207,-74.392,175.193,22.703,153.745
C04801=1083.536,196.958,-74.368,175.191,22.701,153.745
C04802=1083.530,196.709,-74.344,175.188,22.699,153.745
C04803=1083.524,196.460,-74.321,175.186,22.697,153.745
C04804=1083.518,196.211,-74.299,175.183,22.695,153.745
C04805=1083.513,195.962,-74.274,175.181,22.693,153.745
C04806=1083.507,195.713,-74.251,175.179,22.691,153.745
C04807=1083.501,195.464,-74.228,175.176,22.689,153.745
C04808=1083.496,195.215,-74.205,175.174,22.688,153.745
C04809=1083.490,194.967,-74.181,175.171,22.685,153.745
C04810=1083.485,194.718,-74.158,175.169,22.684,153.745
C04811=1083.479,194.469,-74.135,175.166,22.682,153.745
C04812=1083.474,194.220,-74.112,175.164,22.680,153.745
C04813=1083.468,193.971,-74.089,175.162,22.678,153.745
C04814=1083.462,193.723,-74.065,175.158,22.676,153.745
C04815=1083.456,193.474,-74.042,175.156,22.673,153.745
C04816=1083.451,193.225,-74.019,175.153,22.671,153.745
C04817=1083.446,192.976,-73.996,175.151,22.670,153.745
C04818=1083.441,192.728,-73.973,175.149,22.667,153.744
C04819=1083.435,192.479,-73.950,175.146,22.666,153.744
C04820=1083.430,192.229,-73.927,175.144,22.663,153.744
C04821=1083.423,191.951,-73.901,175.141,22.662,153.744
C04822=1083.416,191.672,-73.875,175.139,22.659,153.744
C04823=1083.411,191.394,-73.849,175.136,22.657,153.744
C04824=1083.404,191.114,-73.823,175.133,22.655,153.744
C04825=1083.399,190.865,-73.800,175.131,22.653,153.744
C04826=1083.393,190.616,-73.777,175.128,22.651,153.744
C04827=1083.388,190.367,-73.754,175.126,22.649,153.744
C04828=1083.383,190.119,-73.731,175.124,22.647,153.744
C04829=1083.377,189.870,-73.708,175.121,22.645,153.744
C04830=1083.371,189.621,-73.685,175.119,22.643,153.744
C04831=1083.366,189.372,-73.662,175.116,22.641,153.744
C04832=1083.361,189.123,-73.639,175.114,22.639,153.743
C04833=1083.355,188.874,-73.616,175.112,22.637,153.743
C04834=1083.349,188.625,-73.593,175.109,22.635,153.743
C04835=1083.344,188.377,-73.570,175.107,22.633,153.743
C04836=1083.338,188.128,-73.547,175.104,22.631,153.743
C04837=1083.333,187.879,-73.524,175.102,22.629,153.743
C04838=1083.328,187.630,-73.501,175.100,22.627,153.743
C04839=1083.322,187.381,-73.478,175.097,22.625,153.743
C04840=1083.316,187.132,-73.456,175.095,22.623,153.743
C04841=1083.311,186.883,-73.433,175.092,22.621,153.743
C04842=1083.306,186.635,-73.410,175.090,22.619,153.743
C04843=1083.300,186.386,-73.387,175.087,22.617,153.743
C04844=1083.294,186.137,-73.364,175.085,22.615,153.743
C04845=1083.290,185.888,-73.341,175.083,22.613,153.743
C04846=1083.284,185.639,-73.319,175.080,22.611,153.742
C04847=1083.279,185.390,-73.296,175.078,22.609,153.742
C04848=1083.273,185.141,-73.273,175.076,22.607,153.742
C04849=1083.267,184.892,-73.250,175.073,22.605,153.742
C04850=1083.262,184.642,-73.228,175.071,22.603,153.742
C04851=1083.256,184.395,-73.206,175.068,22.601,153.742
C04852=1083.250,184.146,-73.183,175.066,22.599,153.742
C04853=1083.244,183.897,-73.160,175.063,22.597,153.742
C04854=1083.239,183.647,-73.138,175.061,22.595,153.742
C04855=1083.233,183.398,-73.115,175.058,22.594,153.742
C04856=1083.227,183.150,-73.092,175.056,22.591,153.742
C04857=1083.221,182.900,-73.070,175.054,22.590,153.742
C04858=1083.216,182.651,-73.047,175.051,22.588,153.742
C04859=1083.210,182.403,-73.025,175.049,22.586,153.742
C04860=1083.204,182.154,-73.003,175.047,22.584,153.742
C04861=1083.199,181.905,-72.980,175.045,22.582,153.742
C04862=1083.193,181.656,-72.957,175.042,22.581,153.742
C04863=1083.187,181.407,-72.935,175.040,22.579,153.742
C04864=1083.181,181.158,-72.912,175.038,22.576,153.741
C04865=1083.176,180.910,-72.890,175.035,22.575,153.741
C04866=1083.170,180.660,-72.868,175.033,22.573,153.741
C04867=1083.164,180.412,-72.845,175.030,22.571,153.741
C04868=1083.159,180.162,-72.823,175.028,22.569,153.741
C04869=1083.153,179.913,-72.800,175.025,22.567,153.741
C04870=1083.147,179.665,-72.779,175.023,22.565,153.741
C04871=1083.141,179.416,-72.756,175.021,22.563,153.741
C04872=1083.136,179.167,-72.733,175.018,22.561,153.741
C04873=1083.130,178.918,-72.711,175.016,22.559,153.741
C04874=1083.124,178.670,-72.689,175.013,22.557,153.741
C04875=1083.119,178.420,-72.667,175.012,22.556,153.741
C04876=1083.113,178.171,-72.644,175.009,22.554,153.741
C04877=1083.107,177.922,-72.622,175.007,22.552,153.741
C04878=1083.102,177.673,-72.600,175.004,22.550,153.741
C04879=1083.097,177.424,-72.577,175.002,22.548,153.741
C04880=1083.090,177.175,-72.556,175.000,22.546,153.741
C04881=1083.085,176.926,-72.533,174.997,22.544,153.741
C04882=1083.080,176.677,-72.511,174.995,22.542,153.741
C04883=1083.073,176.429,-72.488,174.992,22.540,153.740
C04884=1083.068,176.179,-72.466,174.990,22.538,153.740
C04885=1083.062,175.901,-72.441,174.988,22.536,153.740
C04886=1083.055,175.621,-72.417,174.985,22.534,153.740
C04887=1083.050,175.343,-72.391,174.983,22.532,153.740
C04888=1083.043,175.063,-72.367,174.979,22.529,153.740
C04889=1083.037,174.814,-72.344,174.978,22.527,153.740
C04890=1083.032,174.565,-72.323,174.976,22.526,153.740
C04891=1083.026,174.316,-72.301,174.973,22.524,153.740
C04892=1083.020,174.067,-72.278,174.971,22.522,153.740
C04893=1083.015,173.819,-72.256,174.968,22.520,153.740
C04894=1083.010,173.569,-72.234,174.966,22.517,153.740
C04895=1083.004,173.321,-72.213,174.964,22.516,153.740
C04896=1082.998,173.072,-72.190,174.961,22.514,153.740
C04897=1082.992,172.822,-72.168,174.959,22.512,153.739
C04898=1082.987,172.574,-72.146,174.957,22.510,153.739
C04899=1082.982,172.324,-72.124,174.955,22.508,153.739
C04900=1082.975,172.075,-72.102,174.952,22.506,153.739
C04901=1082.971,171.827,-72.080,174.950,22.504,153.739
C04902=1082.964,171.577,-72.058,174.948,22.502,153.739
C04903=1082.960,171.329,-72.036,174.945,22.500,153.739
C04904=1082.953,171.079,-72.015,174.943,22.498,153.739
C04905=1082.948,170.831,-71.992,174.940,22.496,153.739
C04906=1082.943,170.582,-71.970,174.939,22.494,153.739
C04907=1082.937,170.333,-71.948,174.937,22.492,153.739
C04908=1082.932,170.084,-71.927,174.934,22.490,153.739
C04909=1082.926,169.834,-71.905,174.932,22.488,153.739
C04910=1082.921,169.586,-71.883,174.929,22.486,153.738
C04911=1082.915,169.336,-71.861,174.927,22.484,153.738
C04912=1082.910,169.088,-71.839,174.925,22.482,153.738
C04913=1082.903,168.839,-71.817,174.923,22.481,153.738
C04914=1082.899,168.590,-71.795,174.921,22.478,153.738
C04915=1082.892,168.341,-71.774,174.918,22.476,153.738
C04916=1082.888,168.092,-71.752,174.916,22.474,153.738
C04917=1082.881,167.843,-71.730,174.914,22.472,153.738
C04918=1082.877,167.594,-71.708,174.911,22.470,153.738
C04919=1082.870,167.345,-71.687,174.910,22.469,153.738
C04920=1082.866,167.096,-71.665,174.907,22.466,153.738
C04921=1082.859,166.847,-71.643,174.905,22.465,153.738
C04922=1082.855,166.598,-71.621,174.903,22.462,153.737
C04923=1082.848,166.349,-71.600,174.900,22.460,153.737
C04924=1082.844,166.100,-71.578,174.898,22.458,153.737
C04925=1082.837,165.851,-71.556,174.897,22.456,153.737
C04926=1082.833,165.602,-71.534,174.894,22.454,153.737
C04927=1082.827,165.353,-71.513,174.892,22.452,153.737
C04928=1082.822,165.104,-71.491,174.889,22.450,153.737
C04929=1082.816,164.855,-71.469,174.887,22.448,153.737
C04930=1082.811,164.606,-71.447,174.885,22.446,153.737
C04931=1082.805,164.358,-71.426,174.883,22.444,153.737
C04932=1082.800,164.107,-71.405,174.881,22.442,153.736
C04933=1082.794,163.859,-71.383,174.878,22.440,153.736
C04934=1082.789,163.609,-71.361,174.876,22.438,153.736
C04935=1082.783,163.361,-71.340,174.874,22.436,153.736
C04936=1082.778,163.112,-71.318,174.872,22.434,153.736
C04937=1082.772,162.863,-71.296,174.870,22.432,153.736
C04938=1082.767,162.614,-71.275,174.867,22.430,153.736
C04939=1082.762,162.364,-71.253,174.865,22.428,153.736
C04940=1082.756,162.116,-71.232,174.863,22.426,153.736
C04941=1082.751,161.867,-71.210,174.860,22.424,153.736
C04942=1082.745,161.618,-71.189,174.859,22.422,153.735
C04943=1082.740,161.369,-71.167,174.856,22.420,153.735
C04944=1082.735,161.119,-71.146,174.854,22.418,153.735
C04945=1082.729,160.871,-71.125,174.852,22.416,153.735
C04946=1082.723,160.622,-71.103,174.849,22.414,153.735
C04947=1082.717,160.373,-71.082,174.848,22.412,153.735
C04948=1082.712,160.124,-71.061,174.846,22.410,153.735
C04949=1082.705,159.844,-71.037,174.843,22.408,153.735
C04950=1082.699,159.565,-71.013,174.841,22.406,153.735
C04951=1082.693,159.285,-70.989,174.838,22.403,153.735
C04952=1082.686,159.006,-70.965,174.835,22.401,153.735
C04953=1082.681,158.756,-70.943,174.834,22.399,153.734
C04954=1082.676,158.507,-70.923,174.831,22.398,153.734
C04955=1082.670,158.259,-70.901,174.829,22.395,153.734
C04956=1082.664,158.010,-70.880,174.827,22.393,153.734
C04957=1082.659,157.761,-70.859,174.824,22.391,153.734
C04958=1082.653,157.511,-70.838,174.823,22.390,153.734
C04959=1082.647,157.263,-70.816,174.820,22.387,153.734
C04960=1082.642,157.014,-70.796,174.818,22.385,153.734
C04961=1082.636,156.764,-70.773,174.816,22.383,153.734
C04962=1082.631,156.516,-70.752,174.814,22.381,153.734
C04963=1082.626,156.267,-70.732,174.812,22.380,153.734
C04964=1082.619,156.017,-70.710,174.809,22.377,153.734
C04965=1082.614,155.768,-70.689,174.807,22.376,153.734
C04966=1082.609,155.520,-70.668,174.806,22.374,153.733
C04967=1082.603,155.270,-70.647,174.803,22.372,153.733
C04968=1082.597,155.021,-70.626,174.801,22.370,153.733
C04969=1082.591,154.772,-70.605,174.798,22.368,153.733
C04970=1082.586,154.523,-70.584,174.797,22.366,153.733
C04971=1082.581,154.274,-70.563,174.795,22.364,153.733
C04972=1082.574,154.025,-70.542,174.792,22.362,153.733
C04973=1082.569,153.776,-70.521,174.790,22.359,153.733
C04974=1082.564,153.527,-70.500,174.788,22.358,153.733
C04975=1082.558,153.277,-70.479,174.786,22.356,153.733
C04976=1082.552,153.029,-70.458,174.784,22.354,153.732
C04977=1082.547,152.780,-70.437,174.781,22.352,153.732
C04978=1082.541,152.531,-70.416,174.780,22.350,153.732
C04979=1082.535,152.281,-70.395,174.777,22.348,153.732
C04980=1082.530,152.032,-70.374,174.775,22.346,153.732
C04981=1082.525,151.784,-70.353,174.773,22.344,153.732
C04982=1082.519,151.534,-70.332,174.771,22.342,153.732
C04983=1082.513,151.285,-70.311,174.769,22.340,153.732
C04984=1082.508,151.036,-70.290,174.767,22.338,153.732
C04985=1082.502,150.787,-70.270,174.764,22.335,153.732
C04986=1082.496,150.538,-70.249,174.763,22.334,153.731
C04987=1082.491,150.289,-70.228,174.760,22.332,153.731
C04988=1082.485,150.040,-70.208,174.758,22.329,153.731
C04989=1082.480,149.791,-70.186,174.756,22.328,153.731
C04990=1082.474,149.542,-70.165,174.754,22.326,153.731
C04991=1082.469,149.293,-70.145,174.752,22.324,153.731
C04992=1082.463,149.044,-70.124,174.750,22.322,153.731
C04993=1082.458,148.795,-70.103,174.748,22.320,153.731
C04994=1082.451,148.545,-70.083,174.746,22.318,153.731
C04995=1082.446,148.296,-70.062,174.743,22.316,153.731
C04996=1082.440,148.048,-70.041,174.741,22.314,153.731
C04997=1082.435,147.799,-70.020,174.739,22.312,153.730
C04998=1082.429,147.549,-69.999,174.737,22.310,153.730
C04999=1082.423,147.300,-69.979,174.735,22.308,153.730
C05000=1082.418,147.051,-69.958,174.733,22.306,153.730
C05001=1082.412,146.802,-69.938,174.731,22.304,153.730
C05002=1082.407,146.553,-69.917,174.729,22.302,153.730
C05003=1082.401,146.304,-69.897,174.726,22.299,153.730
C05004=1082.395,146.055,-69.876,174.725,22.298,153.730
C05005=1082.390,145.806,-69.855,174.722,22.296,153.730
C05006=1082.383,145.557,-69.835,174.720,22.294,153.730
C05007=1082.378,145.307,-69.814,174.719,22.292,153.729
C05008=1082.373,145.058,-69.794,174.716,22.290,153.729
C05009=1082.367,144.809,-69.773,174.714,22.288,153.729
C05010=1082.361,144.560,-69.753,174.712,22.286,153.729
C05011=1082.356,144.311,-69.732,174.710,22.284,153.729
C05012=1082.350,144.061,-69.712,174.708,22.282,153.729
C05013=1082.344,143.782,-69.689,174.705,22.280,153.729
C05014=1082.337,143.503,-69.666,174.703,22.277,153.729
C05015=1082.331,143.222,-69.642,174.701,22.275,153.728
C05016=1082.325,142.943,-69.619,174.699,22.273,153.728
C05017=1082.320,142.694,-69.599,174.696,22.271,153.728
C05018=1082.314,142.445,-69.578,174.695,22.269,153.728
C05019=1082.308,142.196,-69.558,174.692,22.267,153.728
C05020=1082.303,141.947,-69.538,174.690,22.264,153.728
C05021=1082.297,141.697,-69.517,174.689,22.263,153.728
C05022=1082.291,141.448,-69.497,174.686,22.261,153.728
C05023=1082.286,141.199,-69.476,174.684,22.258,153.728
C05024=1082.281,140.950,-69.456,174.682,22.257,153.728
C05025=1082.275,140.701,-69.436,174.680,22.254,153.727
C05026=1082.269,140.452,-69.415,174.678,22.252,153.727
C05027=1082.263,140.203,-69.395,174.677,22.250,153.727
C05028=1082.258,139.954,-69.375,174.674,22.248,153.727
C05029=1082.252,139.705,-69.355,174.672,22.246,153.727
C05030=1082.246,139.456,-69.334,174.670,22.244,153.727
C05031=1082.241,139.206,-69.313,174.668,22.242,153.727
C05032=1082.235,138.958,-69.293,174.666,22.240,153.727
C05033=1082.230,138.708,-69.274,174.664,22.238,153.726
C05034=1082.224,138.459,-69.254,174.662,22.236,153.726
C05035=1082.219,138.210,-69.233,174.660,22.234,153.726
C05036=1082.213,137.961,-69.213,174.658,22.232,153.726
C05037=1082.208,137.712,-69.193,174.656,22.230,153.726
C05038=1082.202,137.463,-69.173,174.653,22.228,153.726
C05039=1082.196,137.214,-69.152,174.652,22.226,153.726
C05040=1082.190,136.964,-69.132,174.650,22.224,153.726
C05041=1082.185,136.715,-69.112,174.647,22.222,153.726
C05042=1082.179,136.466,-69.092,174.646,22.220,153.725
C05043=1082.173,136.217,-69.072,174.644,22.218,153.725
C05044=1082.168,135.968,-69.051,174.641,22.215,153.725
C05045=1082.162,135.719,-69.032,174.640,22.214,153.725
C05046=1082.157,135.469,-69.012,174.637,22.212,153.725
C05047=1082.151,135.221,-68.992,174.635,22.209,153.725
C05048=1082.145,134.972,-68.971,174.634,22.208,153.725
C05049=1082.140,134.722,-68.952,174.631,22.206,153.725
C05050=1082.134,134.473,-68.931,174.629,22.203,153.725
C05051=1082.128,134.224,-68.911,174.628,22.201,153.724
C05052=1082.122,133.975,-68.891,174.625,22.199,153.724
C05053=1082.118,133.726,-68.872,174.624,22.198,153.724
C05054=1082.112,133.477,-68.852,174.622,22.195,153.724
C05055=1082.106,133.228,-68.831,174.619,22.193,153.724
C05056=1082.101,132.978,-68.812,174.618,22.191,153.724
C05057=1082.095,132.729,-68.792,174.615,22.189,153.724
C05058=1082.089,132.480,-68.771,174.613,22.187,153.724
C05059=1082.084,132.231,-68.752,174.612,22.185,153.723
C05060=1082.078,131.982,-68.731,174.610,22.183,153.723
C05061=1082.072,131.733,-68.712,174.607,22.180,153.723
C05062=1082.067,131.484,-68.692,174.606,22.179,153.723
C05063=1082.061,131.235,-68.672,174.603,22.177,153.723
C05064=1082.055,130.985,-68.653,174.602,22.175,153.723
C05065=1082.050,130.736,-68.633,174.600,22.173,153.723
C05066=1082.044,130.487,-68.613,174.597,22.171,153.723
C05067=1082.038,130.238,-68.593,174.596,22.169,153.722
C05068=1082.032,129.989,-68.573,174.594,22.166,153.722
C05069=1082.026,129.740,-68.554,174.592,22.165,153.722
C05070=1082.020,129.491,-68.534,174.590,22.163,153.722
C05071=1082.015,129.241,-68.514,174.587,22.160,153.722
C05072=1082.009,128.992,-68.494,174.586,22.159,153.722
C05073=1082.004,128.743,-68.475,174.584,22.157,153.722
C05074=1081.998,128.494,-68.455,174.581,22.154,153.722
C05075=1081.992,128.245,-68.436,174.580,22.153,153.721
C05076=1081.986,127.996,-68.416,174.578,22.150,153.721
C05077=1081.980,127.716,-68.394,174.575,22.148,153.721
C05078=1081.973,127.435,-68.371,174.573,22.145,153.721
C05079=1081.967,127.155,-68.349,174.572,22.144,153.721
C05080=1081.961,126.876,-68.327,174.570,22.141,153.721
C05081=1081.955,126.626,-68.307,174.567,22.139,153.721
C05082=1081.949,126.377,-68.288,174.565,22.137,153.721
C05083=1081.943,126.128,-68.268,174.563,22.135,153.720
C05084=1081.938,125.879,-68.249,174.561,22.133,153.720
C05085=1081.932,125.631,-68.229,174.560,22.131,153.720
C05086=1081.927,125.381,-68.210,174.557,22.129,153.720
C05087=1081.921,125.132,-68.191,174.555,22.127,153.720
C05088=1081.916,124.883,-68.170,174.554,22.125,153.720
C05089=1081.910,124.633,-68.151,174.551,22.123,153.720
C05090=1081.904,124.384,-68.132,174.550,22.121,153.719
C05091=1081.898,124.135,-68.112,174.548,22.118,153.719
C05092=1081.893,123.886,-68.093,174.545,22.116,153.719
C05093=1081.887,123.636,-68.073,174.544,22.115,153.719
C05094=1081.882,123.388,-68.054,174.542,22.112,153.719
C05095=1081.876,123.139,-68.035,174.540,22.110,153.719
C05096=1081.870,122.889,-68.015,174.538,22.108,153.719
C05097=1081.864,122.640,-67.995,174.537,22.106,153.719
C05098=1081.858,122.391,-67.976,174.534,22.104,153.718
C05099=1081.854,122.141,-67.956,174.532,22.101,153.718
C05100=1081.848,121.892,-67.937,174.531,22.100,153.718
C05101=1081.842,121.644,-67.917,174.528,22.098,153.718
C05102=1081.837,121.394,-67.898,174.527,22.096,153.718
C05103=1081.831,121.145,-67.879,174.525,22.094,153.718
C05104=1081.825,120.895,-67.860,174.523,22.092,153.718
C05105=1081.819,120.647,-67.840,174.521,22.089,153.717
C05106=1081.814,120.397,-67.820,174.519,22.087,153.717
C05107=1081.809,120.148,-67.802,174.517,22.085,153.717
C05108=1081.803,119.899,-67.782,174.515,22.083,153.717
C05109=1081.797,119.650,-67.763,174.514,22.081,153.717
C05110=1081.791,119.401,-67.743,174.511,22.078,153.717
C05111=1081.786,119.151,-67.724,174.510,22.077,153.717
C05112=1081.780,118.903,-67.705,174.508,22.074,153.716
C05113=1081.775,118.653,-67.686,174.505,22.072,153.716
C05114=1081.769,118.404,-67.667,174.504,22.070,153.716
C05115=1081.763,118.154,-67.647,174.502,22.068,153.716
C05116=1081.758,117.906,-67.628,174.500,22.066,153.716
C05117=1081.752,117.657,-67.608,174.498,22.063,153.716
C05118=1081.747,117.407,-67.589,174.497,22.061,153.715
C05119=1081.741,117.158,-67.570,174.494,22.059,153.715
C05120=1081.736,116.909,-67.551,174.493,22.057,153.715
C05121=1081.730,116.660,-67.532,174.491,22.055,153.715
C05122=1081.725,116.410,-67.513,174.489,22.053,153.715
C05123=1081.719,116.161,-67.493,174.487,22.051,153.715
C05124=1081.714,115.912,-67.475,174.485,22.048,153.715
C05125=1081.708,115.663,-67.455,174.484,22.046,153.714
C05126=1081.702,115.413,-67.436,174.481,22.044,153.714
C05127=1081.697,115.164,-67.417,174.480,22.042,153.714
C05128=1081.692,114.915,-67.398,174.478,22.040,153.714
C05129=1081.686,114.666,-67.379,174.476,22.038,153.714
C05130=1081.681,114.417,-67.360,174.474,22.036,153.714
C05131=1081.675,114.167,-67.341,174.472,22.033,153.713
C05132=1081.669,113.918,-67.321,174.470,22.031,153.713
C05133=1081.663,113.669,-67.303,174.468,22.029,153.713
C05134=1081.658,113.420,-67.284,174.467,22.027,153.713
C05135=1081.652,113.171,-67.265,174.464,22.025,153.713
C05136=1081.647,112.921,-67.245,174.463,22.023,153.713
C05137=1081.641,112.672,-67.226,174.461,22.020,153.713
C05138=1081.635,112.423,-67.208,174.459,22.019,153.712
C05139=1081.629,112.174,-67.189,174.457,22.016,153.712
C05140=1081.624,111.924,-67.170,174.456,22.014,153.712
C05141=1081.618,111.645,-67.149,174.454,22.012,153.712
C05142=1081.612,111.364,-67.128,174.451,22.010,153.712
C05143=1081.605,111.085,-67.106,174.449,22.007,153.712
C05144=1081.599,110.805,-67.085,174.447,22.004,153.711
C05145=1081.593,110.555,-67.066,174.446,22.002,153.711
C05146=1081.587,110.307,-67.048,174.443,22.000,153.711
C05147=1081.581,110.057,-67.029,174.442,21.998,153.711
C05148=1081.576,109.808,-67.009,174.440,21.996,153.711
C05149=1081.570,109.559,-66.991,174.438,21.994,153.711
C05150=1081.564,109.309,-66.973,174.436,21.992,153.710
C05151=1081.559,109.060,-66.953,174.435,21.990,153.710
C05152=1081.552,108.811,-66.935,174.432,21.987,153.710
C05153=1081.547,108.562,-66.916,174.431,21.985,153.710
C05154=1081.541,108.313,-66.897,174.429,21.983,153.710
C05155=1081.535,108.063,-66.879,174.427,21.981,153.710
C05156=1081.530,107.814,-66.860,174.425,21.979,153.710
C05157=1081.524,107.565,-66.841,174.424,21.977,153.709
C05158=1081.519,107.316,-66.822,174.421,21.975,153.709
C05159=1081.513,107.066,-66.804,174.420,21.973,153.709
C05160=1081.507,106.817,-66.785,174.418,21.970,153.709
C05161=1081.502,106.568,-66.766,174.416,21.968,153.709
C05162=1081.496,106.319,-66.748,174.414,21.966,153.709
C05163=1081.490,106.069,-66.729,174.413,21.964,153.708
C05164=1081.485,105.821,-66.710,174.411,21.962,153.708
C05165=1081.479,105.571,-66.692,174.409,21.960,153.708
C05166=1081.473,105.321,-66.673,174.407,21.958,153.708
C05167=1081.467,105.073,-66.655,174.406,21.956,153.708
C05168=1081.462,104.823,-66.636,174.403,21.953,153.708
C05169=1081.457,104.574,-66.617,174.402,21.951,153.707
C05170=1081.451,104.325,-66.599,174.400,21.948,153.707
C05171=1081.446,104.076,-66.580,174.399,21.947,153.707
C05172=1081.439,103.827,-66.562,174.396,21.944,153.707
C05173=1081.434,103.576,-66.543,174.395,21.942,153.707
C05174=1081.428,103.328,-66.525,174.393,21.940,153.707
C05175=1081.422,103.079,-66.506,174.391,21.938,153.706
C05176=1081.418,102.829,-66.488,174.389,21.936,153.706
C05177=1081.411,102.580,-66.469,174.388,21.934,153.706
C05178=1081.406,102.331,-66.451,174.385,21.931,153.706
C05179=1081.400,102.082,-66.432,174.384,21.929,153.706
C05180=1081.395,101.832,-66.414,174.382,21.927,153.706
C05181=1081.389,101.583,-66.395,174.381,21.925,153.705
C05182=1081.383,101.333,-66.377,174.378,21.922,153.705
C05183=1081.378,101.085,-66.358,174.377,21.920,153.705
C05184=1081.372,100.835,-66.340,174.375,21.918,153.705
C05185=1081.366,100.586,-66.322,174.373,21.916,153.705
C05186=1081.360,100.337,-66.304,174.371,21.914,153.705
C05187=1081.355,100.088,-66.285,174.370,21.912,153.704
C05188=1081.349,99.838,-66.267,174.367,21.910,153.704
C05189=1081.343,99.589,-66.248,174.366,21.907,153.704
C05190=1081.338,99.340,-66.230,174.364,21.905,153.704
C05191=1081.331,99.090,-66.211,174.363,21.903,153.704
C05192=1081.327,98.841,-66.193,174.360,21.901,153.704
C05193=1081.320,98.592,-66.175,174.359,21.899,153.703
C05194=1081.315,98.343,-66.157,174.357,21.896,153.703
C05195=1081.309,98.093,-66.139,174.355,21.894,153.703
C05196=1081.303,97.845,-66.120,174.353,21.892,153.703
C05197=1081.297,97.595,-66.102,174.352,21.890,153.703
C05198=1081.292,97.346,-66.083,174.350,21.887,153.703
C05199=1081.286,97.096,-66.065,174.348,21.885,153.702
C05200=1081.281,96.847,-66.048,174.347,21.883,153.702
C05201=1081.275,96.598,-66.029,174.345,21.881,153.702
C05202=1081.269,96.349,-66.011,174.343,21.879,153.702
C05203=1081.263,96.099,-65.993,174.341,21.877,153.702
C05204=1081.258,95.850,-65.974,174.340,21.875,153.702
C05205=1081.251,95.570,-65.954,174.338,21.872,153.701
C05206=1081.245,95.291,-65.934,174.335,21.870,153.701
C05207=1081.238,95.011,-65.913,174.333,21.867,153.701
C05208=1081.233,94.730,-65.893,174.332,21.865,153.701
C05209=1081.226,94.481,-65.875,174.330,21.862,153.701
C05210=1081.221,94.232,-65.857,174.329,21.860,153.700
C05211=1081.215,93.983,-65.840,174.326,21.858,153.700
C05212=1081.210,93.734,-65.820,174.325,21.856,153.700
C05213=1081.204,93.485,-65.803,174.323,21.853,153.700
C05214=1081.198,93.235,-65.785,174.321,21.851,153.700
C05215=1081.193,92.986,-65.767,174.319,21.849,153.699
C05216=1081.187,92.736,-65.749,174.318,21.847,153.699
C05217=1081.181,92.487,-65.730,174.317,21.845,153.699
C05218=1081.176,92.238,-65.713,174.314,21.842,153.699
C05219=1081.170,91.988,-65.694,174.313,21.840,153.699
C05220=1081.165,91.739,-65.677,174.311,21.838,153.698
C05221=1081.159,91.490,-65.659,174.309,21.836,153.698
C05222=1081.153,91.241,-65.641,174.307,21.833,153.698
C05223=1081.148,90.992,-65.622,174.306,21.831,153.698
C05224=1081.142,90.742,-65.604,174.304,21.828,153.698
C05225=1081.137,90.493,-65.587,174.302,21.827,153.698
C05226=1081.130,90.243,-65.569,174.300,21.824,153.697
C05227=1081.125,89.994,-65.551,174.299,21.822,153.697
C05228=1081.119,89.745,-65.533,174.297,21.820,153.697
C05229=1081.113,89.495,-65.516,174.295,21.818,153.697
C05230=1081.107,89.246,-65.497,174.294,21.816,153.697
C05231=1081.101,88.997,-65.480,174.292,21.813,153.696
C05232=1081.096,88.748,-65.462,174.290,21.811,153.696
C05233=1081.090,88.499,-65.444,174.288,21.809,153.696
C05234=1081.084,88.249,-65.427,174.287,21.807,153.696
C05235=1081.078,88.000,-65.409,174.285,21.805,153.696
C05236=1081.073,87.751,-65.391,174.283,21.802,153.696
C05237=1081.067,87.502,-65.374,174.282,21.800,153.695
C05238=1081.061,87.252,-65.356,174.280,21.798,153.695
C05239=1081.055,87.003,-65.338,174.278,21.796,153.695
C05240=1081.049,86.753,-65.320,174.276,21.794,153.695
C05241=1081.044,86.504,-65.302,174.275,21.791,153.695
C05242=1081.039,86.255,-65.284,174.274,21.789,153.694
C05243=1081.033,86.005,-65.266,174.271,21.787,153.694
C05244=1081.027,85.756,-65.249,174.270,21.785,153.694
C05245=1081.022,85.507,-65.231,174.268,21.782,153.694
C05246=1081.016,85.257,-65.213,174.267,21.780,153.694
C05247=1081.010,85.008,-65.196,174.264,21.778,153.694
C05248=1081.005,84.759,-65.178,174.263,21.776,153.693
C05249=1080.999,84.509,-65.160,174.262,21.773,153.693
C05250=1080.993,84.260,-65.143,174.260,21.771,153.693
C05251=1080.987,84.011,-65.125,174.258,21.769,153.693
C05252=1080.981,83.762,-65.107,174.256,21.767,153.693
C05253=1080.976,83.512,-65.090,174.255,21.764,153.692
C05254=1080.971,83.263,-65.073,174.253,21.762,153.692
C05255=1080.964,83.013,-65.056,174.251,21.760,153.692
C05256=1080.958,82.764,-65.038,174.250,21.758,153.692
C05257=1080.953,82.515,-65.020,174.248,21.755,153.692
C05258=1080.947,82.266,-65.003,174.246,21.753,153.691
C05259=1080.941,82.017,-64.985,174.244,21.751,153.691
C05260=1080.936,81.767,-64.968,174.243,21.748,153.691
C05261=1080.930,81.518,-64.950,174.242,21.747,153.691
C05262=1080.924,81.268,-64.933,174.239,21.744,153.691
C05263=1080.919,81.019,-64.915,174.238,21.742,153.690
C05264=1080.913,80.770,-64.897,174.236,21.739,153.690
C05265=1080.908,80.521,-64.880,174.235,21.737,153.690
C05266=1080.902,80.271,-64.863,174.233,21.735,153.690
C05267=1080.896,80.022,-64.845,174.231,21.733,153.690
C05268=1080.891,79.773,-64.827,174.230,21.731,153.689
C05269=1080.884,79.493,-64.808,174.228,21.728,153.689
C05270=1080.878,79.213,-64.789,174.226,21.725,153.689
C05271=1080.872,78.933,-64.769,174.224,21.723,153.689
C05272=1080.866,78.653,-64.750,174.222,21.720,153.689
C05273=1080.860,78.404,-64.732,174.220,21.718,153.688
C05274=1080.854,78.155,-64.714,174.219,21.716,153.688
C05275=1080.848,77.906,-64.697,174.218,21.713,153.688
C05276=1080.843,77.656,-64.681,174.215,21.711,153.688
C05277=1080.837,77.407,-64.663,174.214,21.709,153.688
C05278=1080.831,77.157,-64.645,174.212,21.706,153.687
C05279=1080.825,76.908,-64.629,174.211,21.704,153.687
C05280=1080.820,76.659,-64.611,174.209,21.702,153.687
C05281=1080.813,76.409,-64.593,174.207,21.699,153.687
C05282=1080.808,76.160,-64.576,174.206,21.698,153.687
C05283=1080.802,75.911,-64.559,174.204,21.695,153.686
C05284=1080.796,75.662,-64.542,174.202,21.693,153.686
C05285=1080.791,75.412,-64.525,174.201,21.691,153.686
C05286=1080.785,75.163,-64.507,174.199,21.688,153.686
C05287=1080.779,74.913,-64.491,174.197,21.686,153.686
C05288=1080.774,74.664,-64.473,174.196,21.684,153.685
C05289=1080.768,74.415,-64.456,174.194,21.682,153.685
C05290=1080.762,74.165,-64.439,174.193,21.680,153.685
C05291=1080.756,73.916,-64.422,174.191,21.677,153.685
C05292=1080.751,73.666,-64.405,174.189,21.675,153.685
C05293=1080.745,73.417,-64.387,174.188,21.672,153.684
C05294=1080.739,73.168,-64.371,174.186,21.670,153.684
C05295=1080.733,72.918,-64.353,174.185,21.668,153.684
C05296=1080.728,72.669,-64.335,174.182,21.665,153.684
C05297=1080.722,72.420,-64.319,174.181,21.663,153.684
C05298=1080.716,72.171,-64.302,174.180,21.661,153.683
C05299=1080.711,71.921,-64.285,174.178,21.659,153.683
C05300=1080.705,71.672,-64.268,174.176,21.657,153.683
C05301=1080.699,71.422,-64.250,174.175,21.655,153.683
C05302=1080.693,71.173,-64.233,174.173,21.652,153.683
C05303=1080.688,70.924,-64.217,174.172,21.650,153.682
C05304=1080.682,70.675,-64.199,174.170,21.647,153.682
C05305=1080.677,70.425,-64.182,174.168,21.645,153.682
C05306=1080.671,70.176,-64.166,174.167,21.643,153.682
C05307=1080.665,69.927,-64.148,174.165,21.640,153.681
C05308=1080.659,69.677,-64.132,174.163,21.638,153.681
C05309=1080.653,69.427,-64.114,174.161,21.636,153.681
C05310=1080.647,69.178,-64.098,174.160,21.633,153.681
C05311=1080.642,68.929,-64.080,174.159,21.631,153.681
C05312=1080.637,68.679,-64.064,174.156,21.629,153.681
C05313=1080.631,68.430,-64.047,174.155,21.627,153.680
C05314=1080.625,68.181,-64.030,174.154,21.625,153.680
C05315=1080.619,67.932,-64.013,174.152,21.622,153.680
C05316=1080.614,67.682,-63.997,174.151,21.620,153.680
C05317=1080.607,67.433,-63.979,174.149,21.618,153.679
C05318=1080.602,67.183,-63.962,174.147,21.615,153.679
C05319=1080.596,66.934,-63.945,174.146,21.613,153.679
C05320=1080.590,66.685,-63.929,174.144,21.611,153.679
C05321=1080.584,66.435,-63.912,174.142,21.608,153.679
C05322=1080.579,66.186,-63.896,174.141,21.606,153.678
C05323=1080.573,65.937,-63.879,174.139,21.603,153.678
C05324=1080.568,65.687,-63.862,174.138,21.602,153.678
C05325=1080.562,65.438,-63.845,174.136,21.600,153.678
C05326=1080.556,65.189,-63.828,174.134,21.597,153.678
C05327=1080.550,64.939,-63.811,174.133,21.595,153.677
C05328=1080.544,64.689,-63.795,174.132,21.592,153.677
C05329=1080.539,64.440,-63.778,174.130,21.590,153.677
C05330=1080.532,64.191,-63.761,174.128,21.588,153.677
C05331=1080.527,63.941,-63.744,174.126,21.585,153.677
C05332=1080.521,63.692,-63.728,174.125,21.583,153.676
C05333=1080.514,63.412,-63.710,174.123,21.580,153.676
C05334=1080.508,63.133,-63.691,174.121,21.578,153.676
C05335=1080.501,62.853,-63.671,174.119,21.575,153.676
C05336=1080.495,62.573,-63.654,174.118,21.573,153.675
C05337=1080.489,62.323,-63.637,174.116,21.571,153.675
C05338=1080.483,62.074,-63.620,174.115,21.569,153.675
C05339=1080.477,61.825,-63.604,174.112,21.566,153.675
C05340=1080.471,61.575,-63.587,174.111,21.564,153.675
C05341=1080.465,61.326,-63.571,174.110,21.562,153.674
C05342=1080.460,61.076,-63.554,174.108,21.559,153.674
C05343=1080.453,60.826,-63.538,174.107,21.557,153.674
C05344=1080.447,60.578,-63.521,174.105,21.555,153.674
C05345=1080.441,60.328,-63.504,174.103,21.552,153.674
C05346=1080.436,60.079,-63.488,174.102,21.550,153.673
C05347=1080.430,59.829,-63.471,174.100,21.548,153.673
C05348=1080.424,59.580,-63.455,174.098,21.545,153.673
C05349=1080.418,59.331,-63.439,174.097,21.543,153.673
C05350=1080.413,59.081,-63.422,174.096,21.542,153.673
C05351=1080.407,58.832,-63.406,174.094,21.539,153.672
C05352=1080.401,58.582,-63.389,174.092,21.537,153.672
C05353=1080.395,58.333,-63.373,174.091,21.534,153.672
C05354=1080.389,58.084,-63.357,174.089,21.532,153.672
C05355=1080.384,57.835,-63.339,174.088,21.530,153.672
C05356=1080.378,57.585,-63.323,174.086,21.527,153.671
C05357=1080.372,57.336,-63.307,174.084,21.525,153.671
C05358=1080.366,57.086,-63.291,174.083,21.523,153.671
C05359=1080.360,56.837,-63.274,174.082,21.521,153.671
C05360=1080.355,56.587,-63.257,174.080,21.518,153.671
C05361=1080.349,56.338,-63.241,174.078,21.516,153.670
C05362=1080.343,56.089,-63.225,174.077,21.514,153.670
C05363=1080.337,55.839,-63.209,174.075,21.511,153.670
C05364=1080.331,55.590,-63.192,174.074,21.509,153.670
C05365=1080.326,55.340,-63.176,174.072,21.507,153.669
C05366=1080.320,55.090,-63.160,174.070,21.504,153.669
C05367=1080.314,54.841,-63.144,174.069,21.502,153.669
C05368=1080.308,54.592,-63.128,174.068,21.500,153.669
C05369=1080.302,54.342,-63.111,174.066,21.497,153.669
C05370=1080.297,54.094,-63.095,174.064,21.495,153.668
C05371=1080.292,53.844,-63.079,174.063,21.493,153.668
C05372=1080.286,53.595,-63.062,174.061,21.490,153.668
C05373=1080.280,53.345,-63.046,174.060,21.488,153.668
C05374=1080.274,53.096,-63.030,174.059,21.486,153.667
C05375=1080.268,52.847,-63.013,174.056,21.483,153.667
C05376=1080.262,52.597,-62.997,174.055,21.481,153.667
C05377=1080.257,52.347,-62.981,174.054,21.479,153.667
C05378=1080.251,52.098,-62.965,174.052,21.477,153.667
C05379=1080.245,51.848,-62.949,174.050,21.474,153.666
C05380=1080.239,51.599,-62.932,174.049,21.472,153.666
C05381=1080.234,51.350,-62.916,174.047,21.469,153.666
C05382=1080.228,51.101,-62.900,174.046,21.467,153.666
C05383=1080.222,50.851,-62.885,174.045,21.465,153.665
C05384=1080.216,50.602,-62.868,174.042,21.462,153.665
C05385=1080.211,50.352,-62.852,174.041,21.460,153.665
C05386=1080.205,50.103,-62.835,174.040,21.458,153.665
C05387=1080.199,49.853,-62.819,174.038,21.455,153.665
C05388=1080.194,49.604,-62.804,174.036,21.453,153.664
C05389=1080.188,49.355,-62.788,174.035,21.451,153.664
C05390=1080.182,49.105,-62.771,174.033,21.448,153.664
C05391=1080.176,48.856,-62.755,174.032,21.446,153.664
C05392=1080.170,48.606,-62.740,174.031,21.444,153.663
C05393=1080.164,48.357,-62.723,174.029,21.441,153.663
C05394=1080.159,48.108,-62.707,174.027,21.438,153.663
C05395=1080.154,47.858,-62.691,174.026,21.437,153.663
C05396=1080.148,47.608,-62.675,174.025,21.434,153.662
C05397=1080.141,47.328,-62.657,174.023,21.432,153.662
C05398=1080.135,47.048,-62.639,174.021,21.429,153.662
C05399=1080.129,46.768,-62.621,174.020,21.426,153.662
C05400=1080.122,46.489,-62.603,174.018,21.423,153.661
C05401=1080.116,46.239,-62.587,174.016,21.421,153.661
C05402=1080.111,45.989,-62.571,174.015,21.419,153.661
C05403=1080.105,45.740,-62.556,174.013,21.416,153.661
C05404=1080.100,45.491,-62.539,174.012,21.414,153.661
C05405=1080.094,45.241,-62.523,174.011,21.412,153.660
C05406=1080.089,44.991,-62.507,174.008,21.409,153.660
C05407=1080.083,44.743,-62.491,174.007,21.407,153.660
C05408=1080.077,44.493,-62.475,174.006,21.404,153.660
C05409=1080.072,44.243,-62.460,174.004,21.402,153.659
C05410=1080.066,43.994,-62.443,174.003,21.399,153.659
C05411=1080.061,43.745,-62.428,174.001,21.397,153.659
C05412=1080.055,43.495,-62.412,174.000,21.395,153.659
C05413=1080.049,43.246,-62.396,173.998,21.393,153.658
C05414=1080.042,42.996,-62.381,173.997,21.390,153.658
C05415=1080.036,42.747,-62.365,173.996,21.388,153.658
C05416=1080.031,42.498,-62.349,173.993,21.385,153.658
C05417=1080.025,42.248,-62.333,173.992,21.383,153.658
C05418=1080.020,41.998,-62.318,173.991,21.381,153.657
C05419=1080.014,41.749,-62.301,173.989,21.378,153.657
C05420=1080.008,41.499,-62.286,173.988,21.376,153.657
C05421=1080.002,41.251,-62.270,173.986,21.374,153.657
C05422=1079.997,41.001,-62.255,173.985,21.372,153.656
C05423=1079.991,40.751,-62.239,173.983,21.369,153.656
C05424=1079.985,40.501,-62.223,173.982,21.367,153.656
C05425=1079.980,40.253,-62.207,173.980,21.365,153.656
C05426=1079.974,40.003,-62.192,173.978,21.362,153.656
C05427=1079.967,39.754,-62.176,173.977,21.360,153.655
C05428=1079.962,39.505,-62.161,173.976,21.357,153.655
C05429=1079.956,39.255,-62.145,173.974,21.355,153.655
C05430=1079.951,39.005,-62.129,173.973,21.353,153.655
C05431=1079.945,38.755,-62.114,173.971,21.351,153.654
C05432=1079.940,38.507,-62.098,173.970,21.348,153.654
C05433=1079.933,38.257,-62.083,173.968,21.346,153.654
C05434=1079.927,38.008,-62.066,173.967,21.343,153.654
C05435=1079.922,37.758,-62.051,173.965,21.341,153.654
C05436=1079.917,37.508,-62.036,173.963,21.338,153.653
C05437=1079.910,37.259,-62.020,173.962,21.336,153.653
C05438=1079.904,37.009,-62.005,173.961,21.334,153.653
C05439=1079.899,36.761,-61.989,173.960,21.332,153.653
C05440=1079.893,36.511,-61.974,173.958,21.329,153.652
C05441=1079.887,36.261,-61.958,173.956,21.327,153.652
C05442=1079.880,36.012,-61.942,173.955,21.325,153.652
C05443=1079.875,35.763,-61.927,173.953,21.322,153.652
C05444=1079.869,35.513,-61.912,173.952,21.320,153.651
C05445=1079.863,35.264,-61.896,173.950,21.318,153.651
C05446=1079.858,35.014,-61.881,173.949,21.315,153.651
C05447=1079.852,34.765,-61.865,173.947,21.313,153.651
C05448=1079.846,34.515,-61.850,173.946,21.311,153.651
C05449=1079.840,34.266,-61.834,173.945,21.309,153.650
C05450=1079.835,34.016,-61.819,173.943,21.306,153.650
C05451=1079.828,33.767,-61.804,173.941,21.304,153.650
C05452=1079.822,33.517,-61.788,173.940,21.302,153.650
C05453=1079.817,33.268,-61.773,173.939,21.299,153.649
C05454=1079.811,33.018,-61.758,173.937,21.297,153.649
C05455=1079.805,32.768,-61.742,173.935,21.294,153.649
